LIN {X 0,Y 363.878,Z 264.828,A -85,B 0,C 180,E1 -13034.312,E2 -13034.312} C_VEL
LIN {X 0,Y 363.084,Z 274.413,A -85,B 0,C 180,E1 -13035.425,E2 -13035.425} C_VEL
LIN {X 0,Y 362.252,Z 284.208,A -85,B 0,C 180,E1 -13036.823,E2 -13036.823} C_VEL
LIN {X 0,Y 361.616,Z 292.231,A -85,B 0,C 180,E1 -13038.225,E2 -13038.225} C_VEL
LIN {X 0,Y 360.989,Z 300.051,A -85,B 0,C 180,E1 -13039.908,E2 -13039.908} C_VEL
LIN {X 0,Y 360.655,Z 306.321,A -85,B 0,C 180,E1 -13041.596,E2 -13041.596} C_VEL
LIN {X 0,Y 360.41,Z 311.284,A -85,B 0,C 180,E1 -13043.281,E2 -13043.281} C_VEL
LIN {X 0,Y 360.44,Z 315.106,A -85,B 0,C 180,E1 -13044.966,E2 -13044.966} C_VEL
LIN {X 0,Y 360.412,Z 317.873,A -85,B 0,C 180,E1 -13046.646,E2 -13046.646} C_VEL
LIN {X 0,Y 360.513,Z 319.178,A -85,B 0,C 180,E1 -13047.765,E2 -13047.765} C_VEL
LIN {X 0,Y 360.539,Z 320.076,A -85,B 0,C 180,E1 -13048.883,E2 -13048.883} C_VEL
LIN {X 0,Y 360.521,Z 320.55,A -85,B 0,C 180,E1 -13050,E2 -13050} C_VEL
LIN {X 0,Y 360.517,Z 320.6,A -85,B 0,C 180,E1 -13051.117,E2 -13051.117} C_VEL
LIN {X 0,Y 360.427,Z 320.257,A -85,B 0,C 180,E1 -13052.235,E2 -13052.235} C_VEL
LIN {X 0,Y 360.359,Z 319.529,A -85,B 0,C 180,E1 -13053.354,E2 -13053.354} C_VEL
LIN {X 0,Y 360.367,Z 318.397,A -85,B 0,C 180,E1 -13054.474,E2 -13054.474} C_VEL
LIN {X 0,Y 360.407,Z 314.826,A -85,B 0,C 180,E1 -13056.719,E2 -13056.719} C_VEL
LIN {X 0,Y 360.695,Z 310.995,A -85,B 0,C 180,E1 -13058.403,E2 -13058.403} C_VEL
LIN {X 0,Y 361.142,Z 306.058,A -85,B 0,C 180,E1 -13060.087,E2 -13060.087} C_VEL
LIN {X 0,Y 361.814,Z 299.872,A -85,B 0,C 180,E1 -13061.768,E2 -13061.768} C_VEL
LIN {X 0,Y 362.948,Z 292.218,A -85,B 0,C 180,E1 -13063.436,E2 -13063.436} C_VEL
LIN {X 0,Y 363.92,Z 283.963,A -85,B 0,C 180,E1 -13064.899,E2 -13064.899} C_VEL
LIN {X 0,Y 365.228,Z 273.856,A -85,B 0,C 180,E1 -13066.345,E2 -13066.345} C_VEL
LIN {X 0,Y 366.624,Z 263.144,A -85,B 0,C 180,E1 -13067.572,E2 -13067.572} C_VEL
LIN {X 0,Y 367.91,Z 252.779,A -85,B 0,C 180,E1 -13068.516,E2 -13068.516} C_VEL
LIN {X 0,Y 369.141,Z 240.378,A -85,B 0,C 180,E1 -13069.389,E2 -13069.389} C_VEL
LIN {X 0,Y 370.234,Z 227.35,A -85,B 0,C 180,E1 -13070.052,E2 -13070.052} C_VEL
LIN {X 0,Y 370.952,Z 214.539,A -85,B 0,C 180,E1 -13070.481,E2 -13070.481} C_VEL
LIN {X 0,Y 372.245,Z 144.582,A -85,B 0,C 180,E1 -13071.883,E2 -13071.883} C_VEL
LIN {X 0,Y 368.931,Z 123.307,A -85,B 0,C 180,E1 -13072.583,E2 -13072.583} C_VEL
LIN {X 0,Y 365.502,Z 106.451,A -85,B 0,C 180,E1 -13073.214,E2 -13073.214} C_VEL
LIN {X 0,Y 367.15,Z 91.794,A -85,B 0,C 180,E1 -13076.426,E2 -13076.426} C_VEL
LIN {X 0,Y 366.338,Z 86.268,A -85,B 0,C 180,E1 -13077.771,E2 -13077.771} C_VEL
LIN {X 0,Y 363.642,Z 74.544,A -85,B 0,C 180,E1 -13080.807,E2 -13080.807} C_VEL
LIN {X 0,Y 361.899,Z 67.405,A -85,B 0,C 180,E1 -13082.773,E2 -13082.773} C_VEL
LIN {X 0,Y 361.868,Z 67.406,A -85,B 0,C 180,E1 -13085.636,E2 -13085.636} C_VEL
LIN {X 0,Y 361.87,Z 67.408,A -85,B 0,C 180,E1 -13089.027,E2 -13089.027} C_VEL
LIN {X 0,Y 361.835,Z 67.413,A -85,B 0,C 180,E1 -13092.828,E2 -13092.828} C_VEL
LIN {X 0,Y 361.823,Z 67.401,A -85,B 0,C 180,E1 -13095.945,E2 -13095.945} C_VEL
LIN {X 0,Y 361.871,Z 67.406,A -85,B 0,C 180,E1 -13099.237,E2 -13099.237} C_VEL
LIN {X 0,Y 361.867,Z 67.405,A -85,B 0,C 180,E1 -13102.982,E2 -13102.982} C_VEL
LIN {X 0,Y 361.858,Z 67.407,A -85,B 0,C 180,E1 -13106.63,E2 -13106.63} C_VEL
LIN {X 0,Y 361.872,Z 67.404,A -85,B 0,C 180,E1 -13109.672,E2 -13109.672} C_VEL
LIN {X 0,Y 361.952,Z 67.392,A -85,B 0,C 180,E1 -13113.475,E2 -13113.475} C_VEL
LIN {X 0,Y 361.889,Z 67.397,A -85,B 0,C 180,E1 -13117.145,E2 -13117.145} C_VEL
LIN {X 0,Y 361.925,Z 67.399,A -85,B 0,C 180,E1 -13120.725,E2 -13120.725} C_VEL
LIN {X 0,Y 361.943,Z 67.399,A -85,B 0,C 180,E1 -13124.226,E2 -13124.226} C_VEL
LIN {X 0,Y 361.996,Z 67.384,A -85,B 0,C 180,E1 -13126.528,E2 -13126.528} C_VEL
LIN {X 0,Y 362.031,Z 67.39,A -85,B 0,C 180,E1 -13129.938,E2 -13129.938} C_VEL
LIN {X 0,Y 362.158,Z 67.365,A -85,B 0,C 180,E1 -13133.314,E2 -13133.314} C_VEL
LIN {X 0,Y 362.278,Z 67.349,A -85,B 0,C 180,E1 -13137.777,E2 -13137.777} C_VEL
LIN {X 0,Y 362.424,Z 67.341,A -85,B 0,C 180,E1 -13140,E2 -13140} C_VEL
LIN {X 0,Y 362.278,Z 67.348,A -85,B 0,C 180,E1 -13142.224,E2 -13142.224} C_VEL
LIN {X 0,Y 362.146,Z 67.372,A -85,B 0,C 180,E1 -13146.687,E2 -13146.687} C_VEL
LIN {X 0,Y 361.998,Z 67.392,A -85,B 0,C 180,E1 -13150.063,E2 -13150.063} C_VEL
LIN {X 0,Y 361.996,Z 67.389,A -85,B 0,C 180,E1 -13153.899,E2 -13153.899} C_VEL
LIN {X 0,Y 361.926,Z 67.397,A -85,B 0,C 180,E1 -13156.935,E2 -13156.935} C_VEL
LIN {X 0,Y 361.885,Z 67.408,A -85,B 0,C 180,E1 -13160.461,E2 -13160.461} C_VEL
LIN {X 0,Y 361.891,Z 67.406,A -85,B 0,C 180,E1 -13164.113,E2 -13164.113} C_VEL
LIN {X 0,Y 361.863,Z 67.409,A -85,B 0,C 180,E1 -13167.783,E2 -13167.783} C_VEL
LIN {X 0,Y 361.845,Z 67.411,A -85,B 0,C 180,E1 -13171.286,E2 -13171.286} C_VEL
LIN {X 0,Y 361.853,Z 67.412,A -85,B 0,C 180,E1 -13174.281,E2 -13174.281} C_VEL
LIN {X 0,Y 361.859,Z 67.41,A -85,B 0,C 180,E1 -13177.223,E2 -13177.223} C_VEL
LIN {X 0,Y 361.828,Z 67.405,A -85,B 0,C 180,E1 -13180.755,E2 -13180.755} C_VEL
LIN {X 0,Y 361.815,Z 67.414,A -85,B 0,C 180,E1 -13184.369,E2 -13184.369} C_VEL
LIN {X 0,Y 361.83,Z 67.418,A -85,B 0,C 180,E1 -13187.57,E2 -13187.57} C_VEL
LIN {X 0,Y 361.859,Z 67.492,A -85,B 0,C 180,E1 -13191.128,E2 -13191.128} C_VEL
LIN {X 0,Y 362.972,Z 72.191,A -85,B 0,C 180,E1 -13192.606,E2 -13192.606} C_VEL
LIN {X 0,Y 371.01,Z 90.504,A -85,B 0,C 180,E1 -13193.662,E2 -13193.662} C_VEL
LIN {X 0,Y 373.28,Z 96.119,A -85,B 0,C 180,E1 -13193.956,E2 -13193.956} C_VEL
LIN {X 0,Y 371.592,Z 178.35,A -85,B 0,C 180,E1 -13195.596,E2 -13195.596} C_VEL
LIN {X 0,Y 370.967,Z 191.99,A -85,B 0,C 180,E1 -13196.09,E2 -13196.09} C_VEL
LIN {X 0,Y 370.296,Z 204.055,A -85,B 0,C 180,E1 -13196.75,E2 -13196.75} C_VEL
LIN {X 0,Y 369.283,Z 216.174,A -85,B 0,C 180,E1 -13197.639,E2 -13197.639} C_VEL
LIN {X 0,Y 368.162,Z 226.889,A -85,B 0,C 180,E1 -13198.656,E2 -13198.656} C_VEL
LIN {X 0,Y 366.831,Z 237.592,A -85,B 0,C 180,E1 -13199.926,E2 -13199.926} C_VEL
LIN {X 0,Y 365.682,Z 246.772,A -85,B 0,C 180,E1 -13201.284,E2 -13201.284} C_VEL
LIN {X 0,Y 364.549,Z 254.831,A -85,B 0,C 180,E1 -13202.751,E2 -13202.751} C_VEL
LIN {X 0,Y 363.345,Z 262.608,A -85,B 0,C 180,E1 -13204.509,E2 -13204.509} C_VEL
LIN {X 0,Y 362.591,Z 267.841,A -85,B 0,C 180,E1 -13205.982,E2 -13205.982} C_VEL
LIN {X 0,Y 361.848,Z 272.838,A -85,B 0,C 180,E1 -13207.745,E2 -13207.745} C_VEL
LIN {X 0,Y 361.32,Z 276.612,A -85,B 0,C 180,E1 -13209.506,E2 -13209.506} C_VEL
LIN {X 0,Y 360.986,Z 278.531,A -85,B 0,C 180,E1 -13210.673,E2 -13210.673} C_VEL
LIN {X 0,Y 360.598,Z 280.76,A -85,B 0,C 180,E1 -13212.749,E2 -13212.749} C_VEL
LIN {X 0,Y 360.462,Z 281.512,A -85,B 0,C 180,E1 -13214.16,E2 -13214.16} C_VEL
LIN {X 0,Y 360.387,Z 281.658,A -85,B 0,C 180,E1 -13215.315,E2 -13215.315} C_VEL
LIN {X 0,Y 360.421,Z 281.016,A -85,B 0,C 180,E1 -13217.157,E2 -13217.157} C_VEL
LIN {X 0,Y 360.476,Z 279.603,A -85,B 0,C 180,E1 -13218.758,E2 -13218.758} C_VEL
LIN {X 0,Y 360.55,Z 278.064,A -85,B 0,C 180,E1 -13219.897,E2 -13219.897} C_VEL
LIN {X 0,Y 360.842,Z 274.948,A -85,B 0,C 180,E1 -13221.601,E2 -13221.601} C_VEL
LIN {X 0,Y 361.182,Z 270.774,A -85,B 0,C 180,E1 -13223.296,E2 -13223.296} C_VEL
LIN {X 0,Y 361.599,Z 264.43,A -85,B 0,C 180,E1 -13225.262,E2 -13225.262} C_VEL
LIN {X 0,Y 362.197,Z 257.516,A -85,B 0,C 180,E1 -13226.942,E2 -13226.942} C_VEL
LIN {X 0,Y 363.031,Z 248.837,A -85,B 0,C 180,E1 -13228.614,E2 -13228.614} C_VEL
LIN {X 0,Y 363.921,Z 239.937,A -85,B 0,C 180,E1 -13230,E2 -13230} C_VEL
LIN {X 0,Y 364.73,Z 230.191,A -85,B 0,C 180,E1 -13231.243,E2 -13231.243} C_VEL
LIN {X 0,Y 365.603,Z 219.374,A -85,B 0,C 180,E1 -13232.349,E2 -13232.349} C_VEL
LIN {X 0,Y 366.324,Z 207.473,A -85,B 0,C 180,E1 -13233.3,E2 -13233.3} C_VEL
LIN {X 0,Y 366.905,Z 194.367,A -85,B 0,C 180,E1 -13234.085,E2 -13234.085} C_VEL
LIN {X 0,Y 367.322,Z 181.85,A -85,B 0,C 180,E1 -13234.595,E2 -13234.595} C_VEL
LIN {X 0,Y 367.7,Z 164.255,A -85,B 0,C 180,E1 -13235.002,E2 -13235.002} C_VEL
LIN {X 0,Y 368.727,Z 93.086,A -85,B 0,C 180,E1 -13236.387,E2 -13236.387} C_VEL
LIN {X 0,Y 366.646,Z 83.395,A -85,B 0,C 180,E1 -13236.684,E2 -13236.684} C_VEL
LIN {X 0,Y 362.854,Z 71.16,A -85,B 0,C 180,E1 -13237.133,E2 -13237.133} C_VEL
LIN {X 0,Y 362.513,Z 69.324,A -85,B 0,C 180,E1 -13237.64,E2 -13237.64} C_VEL
LIN {X 0,Y 361.863,Z 68,A -85,B 0,C 180,E1 -13238.196,E2 -13238.196} C_VEL
LIN {X 0,Y 360.534,Z 67.575,A -85,B 0,C 180,E1 -13238.93,E2 -13238.93} C_VEL
LIN {X 0,Y 355.937,Z 68.203,A -85,B 0,C 180,E1 -13241.231,E2 -13241.231} C_VEL
LIN {X 0,Y 354.986,Z 68.271,A -85,B 0,C 180,E1 -13242.202,E2 -13242.202} C_VEL
LIN {X 0,Y 354.924,Z 68.276,A -85,B 0,C 180,E1 -13242.53,E2 -13242.53} C_VEL
LIN {X 0,Y 354.925,Z 68.272,A -85,B 0,C 180,E1 -13244.917,E2 -13244.917} C_VEL
LIN {X 0,Y 354.912,Z 68.277,A -85,B 0,C 180,E1 -13248.472,E2 -13248.472} C_VEL
LIN {X 0,Y 354.822,Z 68.289,A -85,B 0,C 180,E1 -13252.107,E2 -13252.107} C_VEL
LIN {X 0,Y 354.903,Z 68.277,A -85,B 0,C 180,E1 -13255.827,E2 -13255.827} C_VEL
LIN {X 0,Y 354.822,Z 68.287,A -85,B 0,C 180,E1 -13259.682,E2 -13259.682} C_VEL
LIN {X 0,Y 354.81,Z 68.29,A -85,B 0,C 180,E1 -13263.702,E2 -13263.702} C_VEL
LIN {X 0,Y 354.806,Z 68.286,A -85,B 0,C 180,E1 -13266.459,E2 -13266.459} C_VEL
LIN {X 0,Y 354.828,Z 68.287,A -85,B 0,C 180,E1 -13269.423,E2 -13269.423} C_VEL
LIN {X 0,Y 354.792,Z 68.288,A -85,B 0,C 180,E1 -13272.867,E2 -13272.867} C_VEL
LIN {X 0,Y 354.784,Z 68.289,A -85,B 0,C 180,E1 -13276.106,E2 -13276.106} C_VEL
LIN {X 0,Y 354.792,Z 68.293,A -85,B 0,C 180,E1 -13279.179,E2 -13279.179} C_VEL
LIN {X 0,Y 354.811,Z 68.285,A -85,B 0,C 180,E1 -13282.402,E2 -13282.402} C_VEL
LIN {X 0,Y 354.816,Z 68.29,A -85,B 0,C 180,E1 -13284.941,E2 -13284.941} C_VEL
LIN {X 0,Y 354.796,Z 68.288,A -85,B 0,C 180,E1 -13288.405,E2 -13288.405} C_VEL
LIN {X 0,Y 354.85,Z 68.28,A -85,B 0,C 180,E1 -13291.618,E2 -13291.618} C_VEL
LIN {X 0,Y 354.902,Z 68.275,A -85,B 0,C 180,E1 -13294.172,E2 -13294.172} C_VEL
LIN {X 0,Y 354.839,Z 68.282,A -85,B 0,C 180,E1 -13297.894,E2 -13297.894} C_VEL
LIN {X 0,Y 354.925,Z 68.272,A -85,B 0,C 180,E1 -13301.891,E2 -13301.891} C_VEL
LIN {X 0,Y 354.946,Z 68.271,A -85,B 0,C 180,E1 -13305.981,E2 -13305.981} C_VEL
LIN {X 0,Y 354.981,Z 68.266,A -85,B 0,C 180,E1 -13309.736,E2 -13309.736} C_VEL
LIN {X 0,Y 355.127,Z 68.246,A -85,B 0,C 180,E1 -13313.18,E2 -13313.18} C_VEL
LIN {X 0,Y 355.245,Z 68.236,A -85,B 0,C 180,E1 -13317.732,E2 -13317.732} C_VEL
LIN {X 0,Y 355.398,Z 68.216,A -85,B 0,C 180,E1 -13320,E2 -13320} C_VEL
LIN {X 0,Y 355.245,Z 68.232,A -85,B 0,C 180,E1 -13322.267,E2 -13322.267} C_VEL
LIN {X 0,Y 355.114,Z 68.248,A -85,B 0,C 180,E1 -13326.819,E2 -13326.819} C_VEL
LIN {X 0,Y 354.958,Z 68.267,A -85,B 0,C 180,E1 -13330.264,E2 -13330.264} C_VEL
LIN {X 0,Y 354.945,Z 68.269,A -85,B 0,C 180,E1 -13334.019,E2 -13334.019} C_VEL
LIN {X 0,Y 354.924,Z 68.271,A -85,B 0,C 180,E1 -13338.108,E2 -13338.108} C_VEL
LIN {X 0,Y 354.817,Z 68.284,A -85,B 0,C 180,E1 -13342.107,E2 -13342.107} C_VEL
LIN {X 0,Y 354.899,Z 68.274,A -85,B 0,C 180,E1 -13345.827,E2 -13345.827} C_VEL
LIN {X 0,Y 354.855,Z 68.279,A -85,B 0,C 180,E1 -13349.678,E2 -13349.678} C_VEL
LIN {X 0,Y 354.808,Z 68.285,A -85,B 0,C 180,E1 -13353.702,E2 -13353.702} C_VEL
LIN {X 0,Y 354.8,Z 68.292,A -85,B 0,C 180,E1 -13356.459,E2 -13356.459} C_VEL
LIN {X 0,Y 354.826,Z 68.283,A -85,B 0,C 180,E1 -13359.423,E2 -13359.423} C_VEL
LIN {X 0,Y 354.789,Z 68.289,A -85,B 0,C 180,E1 -13362.867,E2 -13362.867} C_VEL
LIN {X 0,Y 354.769,Z 68.296,A -85,B 0,C 180,E1 -13366.103,E2 -13366.103} C_VEL
LIN {X 0,Y 354.789,Z 68.288,A -85,B 0,C 180,E1 -13369.179,E2 -13369.179} C_VEL
LIN {X 0,Y 354.809,Z 68.287,A -85,B 0,C 180,E1 -13372.402,E2 -13372.402} C_VEL
LIN {X 0,Y 354.814,Z 68.285,A -85,B 0,C 180,E1 -13374.941,E2 -13374.941} C_VEL
LIN {X 0,Y 354.795,Z 68.288,A -85,B 0,C 180,E1 -13378.405,E2 -13378.405} C_VEL
LIN {X 0,Y 354.882,Z 68.376,A -85,B 0,C 180,E1 -13379.874,E2 -13379.874} C_VEL
LIN {X 0,Y 357.374,Z 80.376,A -85,B 0,C 180,E1 -13382.743,E2 -13382.743} C_VEL
LIN {X 0,Y 358.244,Z 86.354,A -85,B 0,C 180,E1 -13384.119,E2 -13384.119} C_VEL
LIN {X 0,Y 357.097,Z 100.352,A -85,B 0,C 180,E1 -13387.134,E2 -13387.134} C_VEL
LIN {X 0,Y 356.539,Z 106.915,A -85,B 0,C 180,E1 -13388.537,E2 -13388.537} C_VEL
LIN {X 0,Y 361.331,Z 145.067,A -85,B 0,C 180,E1 -13389.568,E2 -13389.568} C_VEL
LIN {X 0,Y 360.23,Z 215.998,A -85,B 0,C 180,E1 -13391,E2 -13391} C_VEL
LIN {X 0,Y 359.668,Z 229.27,A -85,B 0,C 180,E1 -13391.486,E2 -13391.486} C_VEL
LIN {X 0,Y 358.771,Z 242.008,A -85,B 0,C 180,E1 -13392.176,E2 -13392.176} C_VEL
LIN {X 0,Y 357.948,Z 253.353,A -85,B 0,C 180,E1 -13393.018,E2 -13393.018} C_VEL
LIN {X 0,Y 357.002,Z 263.768,A -85,B 0,C 180,E1 -13394.001,E2 -13394.001} C_VEL
LIN {X 0,Y 356.06,Z 274.562,A -85,B 0,C 180,E1 -13395.279,E2 -13395.279} C_VEL
LIN {X 0,Y 355.314,Z 283.359,A -85,B 0,C 180,E1 -13396.561,E2 -13396.561} C_VEL
LIN {X 0,Y 354.6,Z 291.455,A -85,B 0,C 180,E1 -13397.988,E2 -13397.988} C_VEL
LIN {X 0,Y 353.93,Z 299.371,A -85,B 0,C 180,E1 -13399.705,E2 -13399.705} C_VEL
LIN {X 0,Y 353.6,Z 305.7,A -85,B 0,C 180,E1 -13401.427,E2 -13401.427} C_VEL
LIN {X 0,Y 353.352,Z 310.715,A -85,B 0,C 180,E1 -13403.146,E2 -13403.146} C_VEL
LIN {X 0,Y 353.355,Z 314.584,A -85,B 0,C 180,E1 -13404.865,E2 -13404.865} C_VEL
LIN {X 0,Y 353.329,Z 317.395,A -85,B 0,C 180,E1 -13406.579,E2 -13406.579} C_VEL
LIN {X 0,Y 353.415,Z 318.72,A -85,B 0,C 180,E1 -13407.72,E2 -13407.72} C_VEL
LIN {X 0,Y 353.474,Z 319.641,A -85,B 0,C 180,E1 -13408.86,E2 -13408.86} C_VEL
LIN {X 0,Y 353.456,Z 320.152,A -85,B 0,C 180,E1 -13410,E2 -13410} C_VEL
LIN {X 0,Y 353.433,Z 320.225,A -85,B 0,C 180,E1 -13411.139,E2 -13411.139} C_VEL
LIN {X 0,Y 353.275,Z 319.194,A -85,B 0,C 180,E1 -13413.421,E2 -13413.421} C_VEL
LIN {X 0,Y 353.276,Z 318.094,A -85,B 0,C 180,E1 -13414.564,E2 -13414.564} C_VEL
LIN {X 0,Y 353.27,Z 316.242,A -85,B 0,C 180,E1 -13415.897,E2 -13415.897} C_VEL
LIN {X 0,Y 353.528,Z 312.18,A -85,B 0,C 180,E1 -13417.999,E2 -13417.999} C_VEL
LIN {X 0,Y 353.925,Z 307.672,A -85,B 0,C 180,E1 -13419.717,E2 -13419.717} C_VEL
LIN {X 0,Y 354.689,Z 300.891,A -85,B 0,C 180,E1 -13421.718,E2 -13421.718} C_VEL
LIN {X 0,Y 355.832,Z 293.54,A -85,B 0,C 180,E1 -13423.419,E2 -13423.419} C_VEL
LIN {X 0,Y 356.97,Z 284.618,A -85,B 0,C 180,E1 -13425.092,E2 -13425.092} C_VEL
LIN {X 0,Y 358.286,Z 275.092,A -85,B 0,C 180,E1 -13426.524,E2 -13426.524} C_VEL
LIN {X 0,Y 359.71,Z 264.725,A -85,B 0,C 180,E1 -13427.775,E2 -13427.775} C_VEL
LIN {X 0,Y 361.219,Z 253.242,A -85,B 0,C 180,E1 -13428.872,E2 -13428.872} C_VEL
LIN {X 0,Y 362.499,Z 241.208,A -85,B 0,C 180,E1 -13429.759,E2 -13429.759} C_VEL
LIN {X 0,Y 363.682,Z 227.862,A -85,B 0,C 180,E1 -13430.466,E2 -13430.466} C_VEL
LIN {X 0,Y 364.485,Z 214.443,A -85,B 0,C 180,E1 -13430.935,E2 -13430.935} C_VEL
LIN {X 0,Y 365.828,Z 145.241,A -85,B 0,C 180,E1 -13432.347,E2 -13432.347} C_VEL
LIN {X 0,Y 362.406,Z 123.714,A -85,B 0,C 180,E1 -13433.082,E2 -13433.082} C_VEL
LIN {X 0,Y 358.82,Z 106.008,A -85,B 0,C 180,E1 -13433.773,E2 -13433.773} C_VEL
LIN {X 0,Y 360.327,Z 93.124,A -85,B 0,C 180,E1 -13436.654,E2 -13436.654} C_VEL
LIN {X 0,Y 358.869,Z 85.019,A -85,B 0,C 180,E1 -13438.71,E2 -13438.71} C_VEL
LIN {X 0,Y 355.768,Z 71.967,A -85,B 0,C 180,E1 -13442.233,E2 -13442.233} C_VEL
LIN {X 0,Y 354.821,Z 68.289,A -85,B 0,C 180,E1 -13443.3,E2 -13443.3} C_VEL
LIN {X 0,Y 354.798,Z 68.292,A -85,B 0,C 180,E1 -13446.459,E2 -13446.459} C_VEL
LIN {X 0,Y 354.822,Z 68.288,A -85,B 0,C 180,E1 -13449.423,E2 -13449.423} C_VEL
LIN {X 0,Y 354.787,Z 68.291,A -85,B 0,C 180,E1 -13452.867,E2 -13452.867} C_VEL
LIN {X 0,Y 354.773,Z 68.28,A -85,B 0,C 180,E1 -13456.105,E2 -13456.105} C_VEL
LIN {X 0,Y 354.822,Z 68.284,A -85,B 0,C 180,E1 -13459.184,E2 -13459.184} C_VEL
LIN {X 0,Y 354.807,Z 68.282,A -85,B 0,C 180,E1 -13462.402,E2 -13462.402} C_VEL
LIN {X 0,Y 354.81,Z 68.287,A -85,B 0,C 180,E1 -13464.941,E2 -13464.941} C_VEL
LIN {X 0,Y 354.791,Z 68.29,A -85,B 0,C 180,E1 -13468.405,E2 -13468.405} C_VEL
LIN {X 0,Y 354.848,Z 68.282,A -85,B 0,C 180,E1 -13471.619,E2 -13471.619} C_VEL
LIN {X 0,Y 354.897,Z 68.272,A -85,B 0,C 180,E1 -13474.173,E2 -13474.173} C_VEL
LIN {X 0,Y 354.835,Z 68.274,A -85,B 0,C 180,E1 -13477.894,E2 -13477.894} C_VEL
LIN {X 0,Y 354.921,Z 68.266,A -85,B 0,C 180,E1 -13481.891,E2 -13481.891} C_VEL
LIN {X 0,Y 354.94,Z 68.269,A -85,B 0,C 180,E1 -13485.981,E2 -13485.981} C_VEL
LIN {X 0,Y 354.977,Z 68.267,A -85,B 0,C 180,E1 -13489.736,E2 -13489.736} C_VEL
LIN {X 0,Y 355.123,Z 68.241,A -85,B 0,C 180,E1 -13493.181,E2 -13493.181} C_VEL
LIN {X 0,Y 355.241,Z 68.225,A -85,B 0,C 180,E1 -13497.733,E2 -13497.733} C_VEL
LIN {X 0,Y 355.393,Z 68.217,A -85,B 0,C 180,E1 -13500,E2 -13500} C_VEL
LIN {X 0,Y 355.241,Z 68.224,A -85,B 0,C 180,E1 -13502.268,E2 -13502.268} C_VEL
LIN {X 0,Y 355.109,Z 68.249,A -85,B 0,C 180,E1 -13506.82,E2 -13506.82} C_VEL
LIN {X 0,Y 354.954,Z 68.269,A -85,B 0,C 180,E1 -13510.265,E2 -13510.265} C_VEL
LIN {X 0,Y 354.941,Z 68.268,A -85,B 0,C 180,E1 -13514.019,E2 -13514.019} C_VEL
LIN {X 0,Y 354.888,Z 68.271,A -85,B 0,C 180,E1 -13518.093,E2 -13518.093} C_VEL
LIN {X 0,Y 354.817,Z 68.279,A -85,B 0,C 180,E1 -13521.419,E2 -13521.419} C_VEL
LIN {X 0,Y 354.852,Z 68.283,A -85,B 0,C 180,E1 -13524.577,E2 -13524.577} C_VEL
LIN {X 0,Y 354.808,Z 68.288,A -85,B 0,C 180,E1 -13528.385,E2 -13528.385} C_VEL
LIN {X 0,Y 354.786,Z 68.289,A -85,B 0,C 180,E1 -13532.334,E2 -13532.334} C_VEL
LIN {X 0,Y 354.821,Z 68.283,A -85,B 0,C 180,E1 -13535.7,E2 -13535.7} C_VEL
LIN {X 0,Y 354.798,Z 68.293,A -85,B 0,C 180,E1 -13539.419,E2 -13539.419} C_VEL
LIN {X 0,Y 354.785,Z 68.297,A -85,B 0,C 180,E1 -13542.867,E2 -13542.867} C_VEL
LIN {X 0,Y 354.766,Z 68.296,A -85,B 0,C 180,E1 -13546.104,E2 -13546.104} C_VEL
LIN {X 0,Y 354.765,Z 68.295,A -85,B 0,C 180,E1 -13549.177,E2 -13549.177} C_VEL
LIN {X 0,Y 354.816,Z 68.461,A -85,B 0,C 180,E1 -13550.667,E2 -13550.667} C_VEL
LIN {X 0,Y 355.816,Z 72.665,A -85,B 0,C 180,E1 -13552.016,E2 -13552.016} C_VEL
LIN {X 0,Y 364.858,Z 92.844,A -85,B 0,C 180,E1 -13553.226,E2 -13553.226} C_VEL
LIN {X 0,Y 366.995,Z 98.441,A -85,B 0,C 180,E1 -13553.518,E2 -13553.518} C_VEL
LIN {X 0,Y 365.147,Z 179.189,A -85,B 0,C 180,E1 -13555.153,E2 -13555.153} C_VEL
LIN {X 0,Y 364.478,Z 192.945,A -85,B 0,C 180,E1 -13555.667,E2 -13555.667} C_VEL
LIN {X 0,Y 363.747,Z 205.328,A -85,B 0,C 180,E1 -13556.367,E2 -13556.367} C_VEL
LIN {X 0,Y 362.628,Z 217.542,A -85,B 0,C 180,E1 -13557.301,E2 -13557.301} C_VEL
LIN {X 0,Y 361.462,Z 228.075,A -85,B 0,C 180,E1 -13558.334,E2 -13558.334} C_VEL
LIN {X 0,Y 360.035,Z 238.914,A -85,B 0,C 180,E1 -13559.663,E2 -13559.663} C_VEL
LIN {X 0,Y 358.88,Z 247.664,A -85,B 0,C 180,E1 -13561.009,E2 -13561.009} C_VEL
LIN {X 0,Y 357.64,Z 255.855,A -85,B 0,C 180,E1 -13562.551,E2 -13562.551} C_VEL
LIN {X 0,Y 356.435,Z 263.319,A -85,B 0,C 180,E1 -13564.293,E2 -13564.293} C_VEL
LIN {X 0,Y 355.479,Z 269.421,A -85,B 0,C 180,E1 -13566.091,E2 -13566.091} C_VEL
LIN {X 0,Y 354.744,Z 274.153,A -85,B 0,C 180,E1 -13567.889,E2 -13567.889} C_VEL
LIN {X 0,Y 354.382,Z 276.606,A -85,B 0,C 180,E1 -13569.086,E2 -13569.086} C_VEL
LIN {X 0,Y 354.004,Z 278.592,A -85,B 0,C 180,E1 -13570.276,E2 -13570.276} C_VEL
LIN {X 0,Y 353.755,Z 280.127,A -85,B 0,C 180,E1 -13571.466,E2 -13571.466} C_VEL
LIN {X 0,Y 353.539,Z 281.176,A -85,B 0,C 180,E1 -13572.652,E2 -13572.652} C_VEL
LIN {X 0,Y 353.408,Z 281.814,A -85,B 0,C 180,E1 -13573.835,E2 -13573.835} C_VEL
LIN {X 0,Y 353.329,Z 282.052,A -85,B 0,C 180,E1 -13575.015,E2 -13575.015} C_VEL
LIN {X 0,Y 353.342,Z 281.431,A -85,B 0,C 180,E1 -13577.065,E2 -13577.065} C_VEL
LIN {X 0,Y 353.39,Z 280.199,A -85,B 0,C 180,E1 -13578.529,E2 -13578.529} C_VEL
LIN {X 0,Y 353.437,Z 278.774,A -85,B 0,C 180,E1 -13579.691,E2 -13579.691} C_VEL
LIN {X 0,Y 353.736,Z 275.777,A -85,B 0,C 180,E1 -13581.431,E2 -13581.431} C_VEL
LIN {X 0,Y 354.081,Z 271.736,A -85,B 0,C 180,E1 -13583.161,E2 -13583.161} C_VEL
LIN {X 0,Y 354.495,Z 265.54,A -85,B 0,C 180,E1 -13585.167,E2 -13585.167} C_VEL
LIN {X 0,Y 355.089,Z 258.789,A -85,B 0,C 180,E1 -13586.88,E2 -13586.88} C_VEL
LIN {X 0,Y 355.939,Z 250.388,A -85,B 0,C 180,E1 -13588.586,E2 -13588.586} C_VEL
LIN {X 0,Y 356.795,Z 241.73,A -85,B 0,C 180,E1 -13590,E2 -13590} C_VEL
LIN {X 0,Y 357.743,Z 231.09,A -85,B 0,C 180,E1 -13591.408,E2 -13591.408} C_VEL
LIN {X 0,Y 358.694,Z 220.019,A -85,B 0,C 180,E1 -13592.572,E2 -13592.572} C_VEL
LIN {X 0,Y 359.412,Z 208.174,A -85,B 0,C 180,E1 -13593.543,E2 -13593.543} C_VEL
LIN {X 0,Y 360.046,Z 194.964,A -85,B 0,C 180,E1 -13594.353,E2 -13594.353} C_VEL
LIN {X 0,Y 360.48,Z 181.966,A -85,B 0,C 180,E1 -13594.893,E2 -13594.893} C_VEL
LIN {X 0,Y 360.875,Z 164.179,A -85,B 0,C 180,E1 -13595.308,E2 -13595.308} C_VEL
LIN {X 0,Y 361.903,Z 93.961,A -85,B 0,C 180,E1 -13596.701,E2 -13596.701} C_VEL
LIN {X 0,Y 359.981,Z 85.067,A -85,B 0,C 180,E1 -13596.981,E2 -13596.981} C_VEL
LIN {X 0,Y 355.719,Z 71.491,A -85,B 0,C 180,E1 -13597.504,E2 -13597.504} C_VEL
LIN {X 0,Y 355.112,Z 68.253,A -85,B 0,C 180,E1 -13598.444,E2 -13598.444} C_VEL
LIN {X 0,Y 354.924,Z 68.276,A -85,B 0,C 180,E1 -13602.53,E2 -13602.53} C_VEL
LIN {X 0,Y 354.278,Z 68.363,A -85,B 0,C 180,E1 -13603.477,E2 -13603.477} C_VEL
LIN {X 0,Y 351.382,Z 68.721,A -85,B 0,C 180,E1 -13605.015,E2 -13605.015} C_VEL
LIN {X 0,Y 348.937,Z 69.022,A -85,B 0,C 180,E1 -13606.261,E2 -13606.261} C_VEL
LIN {X 0,Y 347.925,Z 69.143,A -85,B 0,C 180,E1 -13607.225,E2 -13607.225} C_VEL
LIN {X 0,Y 347.864,Z 69.151,A -85,B 0,C 180,E1 -13607.552,E2 -13607.552} C_VEL
LIN {X 0,Y 347.786,Z 69.16,A -85,B 0,C 180,E1 -13611.331,E2 -13611.331} C_VEL
LIN {X 0,Y 347.816,Z 69.156,A -85,B 0,C 180,E1 -13615.109,E2 -13615.109} C_VEL
LIN {X 0,Y 347.813,Z 69.16,A -85,B 0,C 180,E1 -13617.694,E2 -13617.694} C_VEL
LIN {X 0,Y 347.754,Z 69.166,A -85,B 0,C 180,E1 -13620.348,E2 -13620.348} C_VEL
LIN {X 0,Y 347.753,Z 69.167,A -85,B 0,C 180,E1 -13624.044,E2 -13624.044} C_VEL
LIN {X 0,Y 347.77,Z 69.165,A -85,B 0,C 180,E1 -13627.32,E2 -13627.32} C_VEL
LIN {X 0,Y 347.737,Z 69.167,A -85,B 0,C 180,E1 -13630.297,E2 -13630.297} C_VEL
LIN {X 0,Y 347.727,Z 69.173,A -85,B 0,C 180,E1 -13633.408,E2 -13633.408} C_VEL
LIN {X 0,Y 347.731,Z 69.168,A -85,B 0,C 180,E1 -13636.686,E2 -13636.686} C_VEL
LIN {X 0,Y 347.751,Z 69.164,A -85,B 0,C 180,E1 -13640.173,E2 -13640.173} C_VEL
LIN {X 0,Y 347.765,Z 69.165,A -85,B 0,C 180,E1 -13642.679,E2 -13642.679} C_VEL
LIN {X 0,Y 347.752,Z 69.164,A -85,B 0,C 180,E1 -13645.956,E2 -13645.956} C_VEL
LIN {X 0,Y 347.753,Z 69.164,A -85,B 0,C 180,E1 -13649.652,E2 -13649.652} C_VEL
LIN {X 0,Y 347.834,Z 69.154,A -85,B 0,C 180,E1 -13653.607,E2 -13653.607} C_VEL
LIN {X 0,Y 347.793,Z 69.161,A -85,B 0,C 180,E1 -13656.162,E2 -13656.162} C_VEL
LIN {X 0,Y 347.816,Z 69.157,A -85,B 0,C 180,E1 -13659.909,E2 -13659.909} C_VEL
LIN {X 0,Y 347.869,Z 69.155,A -85,B 0,C 180,E1 -13662.359,E2 -13662.359} C_VEL
LIN {X 0,Y 347.9,Z 69.149,A -85,B 0,C 180,E1 -13665.971,E2 -13665.971} C_VEL
LIN {X 0,Y 347.931,Z 69.143,A -85,B 0,C 180,E1 -13669.525,E2 -13669.525} C_VEL
LIN {X 0,Y 348.093,Z 69.122,A -85,B 0,C 180,E1 -13673.042,E2 -13673.042} C_VEL
LIN {X 0,Y 348.208,Z 69.112,A -85,B 0,C 180,E1 -13677.686,E2 -13677.686} C_VEL
LIN {X 0,Y 348.347,Z 69.094,A -85,B 0,C 180,E1 -13680,E2 -13680} C_VEL
LIN {X 0,Y 348.208,Z 69.108,A -85,B 0,C 180,E1 -13682.313,E2 -13682.313} C_VEL
LIN {X 0,Y 348.079,Z 69.125,A -85,B 0,C 180,E1 -13686.958,E2 -13686.958} C_VEL
LIN {X 0,Y 347.899,Z 69.146,A -85,B 0,C 180,E1 -13690.475,E2 -13690.475} C_VEL
LIN {X 0,Y 347.901,Z 69.146,A -85,B 0,C 180,E1 -13694.15,E2 -13694.15} C_VEL
LIN {X 0,Y 347.893,Z 69.147,A -85,B 0,C 180,E1 -13698.29,E2 -13698.29} C_VEL
LIN {X 0,Y 347.769,Z 69.163,A -85,B 0,C 180,E1 -13701.626,E2 -13701.626} C_VEL
LIN {X 0,Y 347.813,Z 69.161,A -85,B 0,C 180,E1 -13705.108,E2 -13705.108} C_VEL
LIN {X 0,Y 347.811,Z 69.157,A -85,B 0,C 180,E1 -13707.694,E2 -13707.694} C_VEL
LIN {X 0,Y 347.766,Z 69.165,A -85,B 0,C 180,E1 -13710.346,E2 -13710.346} C_VEL
LIN {X 0,Y 347.746,Z 69.17,A -85,B 0,C 180,E1 -13714.464,E2 -13714.464} C_VEL
LIN {X 0,Y 347.775,Z 69.163,A -85,B 0,C 180,E1 -13717.988,E2 -13717.988} C_VEL
LIN {X 0,Y 347.752,Z 69.166,A -85,B 0,C 180,E1 -13721.83,E2 -13721.83} C_VEL
LIN {X 0,Y 347.707,Z 69.17,A -85,B 0,C 180,E1 -13725.026,E2 -13725.026} C_VEL
LIN {X 0,Y 347.752,Z 69.167,A -85,B 0,C 180,E1 -13728.397,E2 -13728.397} C_VEL
LIN {X 0,Y 347.775,Z 69.167,A -85,B 0,C 180,E1 -13732.011,E2 -13732.011} C_VEL
LIN {X 0,Y 347.746,Z 69.168,A -85,B 0,C 180,E1 -13735.536,E2 -13735.536} C_VEL
LIN {X 0,Y 347.848,Z 69.323,A -85,B 0,C 180,E1 -13739.619,E2 -13739.619} C_VEL
LIN {X 0,Y 350.306,Z 81.191,A -85,B 0,C 180,E1 -13742.52,E2 -13742.52} C_VEL
LIN {X 0,Y 351.24,Z 86.967,A -85,B 0,C 180,E1 -13743.883,E2 -13743.883} C_VEL
LIN {X 0,Y 350.393,Z 98.157,A -85,B 0,C 180,E1 -13746.35,E2 -13746.35} C_VEL
LIN {X 0,Y 349.601,Z 106.602,A -85,B 0,C 180,E1 -13748.191,E2 -13748.191} C_VEL
LIN {X 0,Y 354.508,Z 145.666,A -85,B 0,C 180,E1 -13749.259,E2 -13749.259} C_VEL
LIN {X 0,Y 353.401,Z 215.496,A -85,B 0,C 180,E1 -13750.693,E2 -13750.693} C_VEL
LIN {X 0,Y 352.853,Z 228.044,A -85,B 0,C 180,E1 -13751.153,E2 -13751.153} C_VEL
LIN {X 0,Y 351.892,Z 241.574,A -85,B 0,C 180,E1 -13751.891,E2 -13751.891} C_VEL
LIN {X 0,Y 350.978,Z 253.74,A -85,B 0,C 180,E1 -13752.821,E2 -13752.821} C_VEL
LIN {X 0,Y 350.011,Z 264.014,A -85,B 0,C 180,E1 -13753.823,E2 -13753.823} C_VEL
LIN {X 0,Y 349.011,Z 274.84,A -85,B 0,C 180,E1 -13755.144,E2 -13755.144} C_VEL
LIN {X 0,Y 348.169,Z 284.302,A -85,B 0,C 180,E1 -13756.577,E2 -13756.577} C_VEL
LIN {X 0,Y 347.358,Z 293.536,A -85,B 0,C 180,E1 -13758.327,E2 -13758.327} C_VEL
LIN {X 0,Y 346.753,Z 300.964,A -85,B 0,C 180,E1 -13760.079,E2 -13760.079} C_VEL
LIN {X 0,Y 346.46,Z 306.918,A -85,B 0,C 180,E1 -13761.836,E2 -13761.836} C_VEL
LIN {X 0,Y 346.238,Z 311.727,A -85,B 0,C 180,E1 -13763.648,E2 -13763.648} C_VEL
LIN {X 0,Y 346.302,Z 315.14,A -85,B 0,C 180,E1 -13765.343,E2 -13765.343} C_VEL
LIN {X 0,Y 346.249,Z 316.917,A -85,B 0,C 180,E1 -13766.509,E2 -13766.509} C_VEL
LIN {X 0,Y 346.317,Z 318.262,A -85,B 0,C 180,E1 -13767.673,E2 -13767.673} C_VEL
LIN {X 0,Y 346.41,Z 319.206,A -85,B 0,C 180,E1 -13768.837,E2 -13768.837} C_VEL
LIN {X 0,Y 346.392,Z 319.746,A -85,B 0,C 180,E1 -13770,E2 -13770} C_VEL
LIN {X 0,Y 346.35,Z 319.849,A -85,B 0,C 180,E1 -13771.162,E2 -13771.162} C_VEL
LIN {X 0,Y 346.193,Z 318.858,A -85,B 0,C 180,E1 -13773.491,E2 -13773.491} C_VEL
LIN {X 0,Y 346.188,Z 317.783,A -85,B 0,C 180,E1 -13774.657,E2 -13774.657} C_VEL
LIN {X 0,Y 346.197,Z 316.178,A -85,B 0,C 180,E1 -13775.884,E2 -13775.884} C_VEL
LIN {X 0,Y 346.48,Z 311.951,A -85,B 0,C 180,E1 -13778.162,E2 -13778.162} C_VEL
LIN {X 0,Y 346.894,Z 307.492,A -85,B 0,C 180,E1 -13779.916,E2 -13779.916} C_VEL
LIN {X 0,Y 347.709,Z 300.798,A -85,B 0,C 180,E1 -13781.956,E2 -13781.956} C_VEL
LIN {X 0,Y 348.911,Z 293.517,A -85,B 0,C 180,E1 -13783.69,E2 -13783.69} C_VEL
LIN {X 0,Y 350.02,Z 285.272,A -85,B 0,C 180,E1 -13785.291,E2 -13785.291} C_VEL
LIN {X 0,Y 351.478,Z 275.287,A -85,B 0,C 180,E1 -13786.854,E2 -13786.854} C_VEL
LIN {X 0,Y 352.982,Z 265.045,A -85,B 0,C 180,E1 -13788.125,E2 -13788.125} C_VEL
LIN {X 0,Y 354.526,Z 253.723,A -85,B 0,C 180,E1 -13789.242,E2 -13789.242} C_VEL
LIN {X 0,Y 355.866,Z 241.993,A -85,B 0,C 180,E1 -13790.143,E2 -13790.143} C_VEL
LIN {X 0,Y 357.074,Z 229.144,A -85,B 0,C 180,E1 -13790.862,E2 -13790.862} C_VEL
LIN {X 0,Y 358,Z 215.468,A -85,B 0,C 180,E1 -13791.371,E2 -13791.371} C_VEL
LIN {X 0,Y 359.49,Z 146.357,A -85,B 0,C 180,E1 -13792.814,E2 -13792.814} C_VEL
LIN {X 0,Y 355.918,Z 124.025,A -85,B 0,C 180,E1 -13793.602,E2 -13793.602} C_VEL
LIN {X 0,Y 352.14,Z 105.526,A -85,B 0,C 180,E1 -13794.364,E2 -13794.364} C_VEL
LIN {X 0,Y 353.472,Z 95.117,A -85,B 0,C 180,E1 -13796.739,E2 -13796.739} C_VEL
LIN {X 0,Y 352.461,Z 88.724,A -85,B 0,C 180,E1 -13798.377,E2 -13798.377} C_VEL
LIN {X 0,Y 349.795,Z 77.298,A -85,B 0,C 180,E1 -13801.492,E2 -13801.492} C_VEL
LIN {X 0,Y 347.771,Z 69.172,A -85,B 0,C 180,E1 -13803.83,E2 -13803.83} C_VEL
LIN {X 0,Y 347.762,Z 69.166,A -85,B 0,C 180,E1 -13807.32,E2 -13807.32} C_VEL
LIN {X 0,Y 347.731,Z 69.17,A -85,B 0,C 180,E1 -13810.296,E2 -13810.296} C_VEL
LIN {X 0,Y 347.721,Z 69.174,A -85,B 0,C 180,E1 -13813.408,E2 -13813.408} C_VEL
LIN {X 0,Y 347.744,Z 69.161,A -85,B 0,C 180,E1 -13816.682,E2 -13816.682} C_VEL
LIN {X 0,Y 347.756,Z 69.166,A -85,B 0,C 180,E1 -13820.171,E2 -13820.171} C_VEL
LIN {X 0,Y 347.769,Z 69.165,A -85,B 0,C 180,E1 -13823.934,E2 -13823.934} C_VEL
LIN {X 0,Y 347.74,Z 69.168,A -85,B 0,C 180,E1 -13826.929,E2 -13826.929} C_VEL
LIN {X 0,Y 347.803,Z 69.163,A -85,B 0,C 180,E1 -13830.99,E2 -13830.99} C_VEL
LIN {X 0,Y 347.829,Z 69.151,A -85,B 0,C 180,E1 -13833.608,E2 -13833.608} C_VEL
LIN {X 0,Y 347.786,Z 69.162,A -85,B 0,C 180,E1 -13836.162,E2 -13836.162} C_VEL
LIN {X 0,Y 347.825,Z 69.157,A -85,B 0,C 180,E1 -13839.91,E2 -13839.91} C_VEL
LIN {X 0,Y 347.864,Z 69.144,A -85,B 0,C 180,E1 -13842.359,E2 -13842.359} C_VEL
LIN {X 0,Y 347.895,Z 69.147,A -85,B 0,C 180,E1 -13845.971,E2 -13845.971} C_VEL
LIN {X 0,Y 347.927,Z 69.144,A -85,B 0,C 180,E1 -13849.526,E2 -13849.526} C_VEL
LIN {X 0,Y 348.089,Z 69.117,A -85,B 0,C 180,E1 -13853.042,E2 -13853.042} C_VEL
LIN {X 0,Y 348.203,Z 69.101,A -85,B 0,C 180,E1 -13857.687,E2 -13857.687} C_VEL
LIN {X 0,Y 348.342,Z 69.095,A -85,B 0,C 180,E1 -13860,E2 -13860} C_VEL
LIN {X 0,Y 348.203,Z 69.1,A -85,B 0,C 180,E1 -13862.314,E2 -13862.314} C_VEL
LIN {X 0,Y 348.075,Z 69.124,A -85,B 0,C 180,E1 -13866.959,E2 -13866.959} C_VEL
LIN {X 0,Y 347.894,Z 69.148,A -85,B 0,C 180,E1 -13870.476,E2 -13870.476} C_VEL
LIN {X 0,Y 347.896,Z 69.145,A -85,B 0,C 180,E1 -13874.15,E2 -13874.15} C_VEL
LIN {X 0,Y 347.827,Z 69.151,A -85,B 0,C 180,E1 -13878.26,E2 -13878.26} C_VEL
LIN {X 0,Y 347.766,Z 69.156,A -85,B 0,C 180,E1 -13881.627,E2 -13881.627} C_VEL
LIN {X 0,Y 347.791,Z 69.156,A -85,B 0,C 180,E1 -13885.111,E2 -13885.111} C_VEL
LIN {X 0,Y 347.755,Z 69.161,A -85,B 0,C 180,E1 -13889.015,E2 -13889.015} C_VEL
LIN {X 0,Y 347.732,Z 69.169,A -85,B 0,C 180,E1 -13893.073,E2 -13893.073} C_VEL
LIN {X 0,Y 347.769,Z 69.165,A -85,B 0,C 180,E1 -13896.066,E2 -13896.066} C_VEL
LIN {X 0,Y 347.73,Z 69.174,A -85,B 0,C 180,E1 -13898.796,E2 -13898.796} C_VEL
LIN {X 0,Y 347.746,Z 69.161,A -85,B 0,C 180,E1 -13901.832,E2 -13901.832} C_VEL
LIN {X 0,Y 347.704,Z 69.169,A -85,B 0,C 180,E1 -13905.028,E2 -13905.028} C_VEL
LIN {X 0,Y 347.741,Z 69.171,A -85,B 0,C 180,E1 -13908.4,E2 -13908.4} C_VEL
LIN {X 0,Y 347.721,Z 69.219,A -85,B 0,C 180,E1 -13910.1,E2 -13910.1} C_VEL
LIN {X 0,Y 348.694,Z 73.239,A -85,B 0,C 180,E1 -13911.389,E2 -13911.389} C_VEL
LIN {X 0,Y 357.548,Z 92.446,A -85,B 0,C 180,E1 -13912.612,E2 -13912.612} C_VEL
LIN {X 0,Y 360.625,Z 99.914,A -85,B 0,C 180,E1 -13913.038,E2 -13913.038} C_VEL
LIN {X 0,Y 358.776,Z 178.778,A -85,B 0,C 180,E1 -13914.657,E2 -13914.657} C_VEL
LIN {X 0,Y 358.092,Z 192.005,A -85,B 0,C 180,E1 -13915.138,E2 -13915.138} C_VEL
LIN {X 0,Y 357.354,Z 204.58,A -85,B 0,C 180,E1 -13915.841,E2 -13915.841} C_VEL
LIN {X 0,Y 356.356,Z 215.514,A -85,B 0,C 180,E1 -13916.651,E2 -13916.651} C_VEL
LIN {X 0,Y 355.101,Z 226.551,A -85,B 0,C 180,E1 -13917.699,E2 -13917.699} C_VEL
LIN {X 0,Y 353.619,Z 237.731,A -85,B 0,C 180,E1 -13919.053,E2 -13919.053} C_VEL
LIN {X 0,Y 352.27,Z 246.764,A -85,B 0,C 180,E1 -13920.411,E2 -13920.411} C_VEL
LIN {X 0,Y 350.923,Z 255.815,A -85,B 0,C 180,E1 -13922.11,E2 -13922.11} C_VEL
LIN {X 0,Y 349.706,Z 262.89,A -85,B 0,C 180,E1 -13923.761,E2 -13923.761} C_VEL
LIN {X 0,Y 348.667,Z 269.178,A -85,B 0,C 180,E1 -13925.603,E2 -13925.603} C_VEL
LIN {X 0,Y 347.838,Z 274.028,A -85,B 0,C 180,E1 -13927.426,E2 -13927.426} C_VEL
LIN {X 0,Y 347.251,Z 277.694,A -85,B 0,C 180,E1 -13929.257,E2 -13929.257} C_VEL
LIN {X 0,Y 346.76,Z 280.263,A -85,B 0,C 180,E1 -13931.078,E2 -13931.078} C_VEL
LIN {X 0,Y 346.479,Z 281.517,A -85,B 0,C 180,E1 -13932.432,E2 -13932.432} C_VEL
LIN {X 0,Y 346.249,Z 282.414,A -85,B 0,C 180,E1 -13934.701,E2 -13934.701} C_VEL
LIN {X 0,Y 346.269,Z 281.848,A -85,B 0,C 180,E1 -13936.966,E2 -13936.966} C_VEL
LIN {X 0,Y 346.279,Z 280.794,A -85,B 0,C 180,E1 -13938.291,E2 -13938.291} C_VEL
LIN {X 0,Y 346.328,Z 279.437,A -85,B 0,C 180,E1 -13939.477,E2 -13939.477} C_VEL
LIN {X 0,Y 346.615,Z 276.557,A -85,B 0,C 180,E1 -13941.254,E2 -13941.254} C_VEL
LIN {X 0,Y 346.947,Z 272.647,A -85,B 0,C 180,E1 -13943.019,E2 -13943.019} C_VEL
LIN {X 0,Y 347.294,Z 267.616,A -85,B 0,C 180,E1 -13944.776,E2 -13944.776} C_VEL
LIN {X 0,Y 347.859,Z 261.286,A -85,B 0,C 180,E1 -13946.526,E2 -13946.526} C_VEL
LIN {X 0,Y 348.703,Z 253.338,A -85,B 0,C 180,E1 -13948.268,E2 -13948.268} C_VEL
LIN {X 0,Y 349.494,Z 245.258,A -85,B 0,C 180,E1 -13949.712,E2 -13949.712} C_VEL
LIN {X 0,Y 350.475,Z 235.394,A -85,B 0,C 180,E1 -13951.149,E2 -13951.149} C_VEL
LIN {X 0,Y 351.333,Z 225.708,A -85,B 0,C 180,E1 -13952.293,E2 -13952.293} C_VEL
LIN {X 0,Y 352.272,Z 213.486,A -85,B 0,C 180,E1 -13953.432,E2 -13953.432} C_VEL
LIN {X 0,Y 352.987,Z 200.862,A -85,B 0,C 180,E1 -13954.328,E2 -13954.328} C_VEL
LIN {X 0,Y 353.489,Z 187.717,A -85,B 0,C 180,E1 -13954.99,E2 -13954.99} C_VEL
LIN {X 0,Y 353.896,Z 174.188,A -85,B 0,C 180,E1 -13955.413,E2 -13955.413} C_VEL
LIN {X 0,Y 355.227,Z 95.348,A -85,B 0,C 180,E1 -13957.005,E2 -13957.005} C_VEL
LIN {X 0,Y 353.361,Z 86.985,A -85,B 0,C 180,E1 -13957.277,E2 -13957.277} C_VEL
LIN {X 0,Y 348.591,Z 71.835,A -85,B 0,C 180,E1 -13957.881,E2 -13957.881} C_VEL
LIN {X 0,Y 348.023,Z 69.136,A -85,B 0,C 180,E1 -13958.727,E2 -13958.727} C_VEL
LIN {X 0,Y 347.895,Z 69.149,A -85,B 0,C 180,E1 -13962.84,E2 -13962.84} C_VEL
LIN {X 0,Y 347.845,Z 69.158,A -85,B 0,C 180,E1 -13966.431,E2 -13966.431} C_VEL
LIN {X 0,Y 347.864,Z 69.151,A -85,B 0,C 180,E1 -13967.552,E2 -13967.552} C_VEL
LIN {X 0,Y 347.236,Z 69.233,A -85,B 0,C 180,E1 -13968.518,E2 -13968.518} C_VEL
LIN {X 0,Y 344.328,Z 69.595,A -85,B 0,C 180,E1 -13970.087,E2 -13970.087} C_VEL
LIN {X 0,Y 341.84,Z 69.902,A -85,B 0,C 180,E1 -13971.357,E2 -13971.357} C_VEL
LIN {X 0,Y 340.785,Z 70.036,A -85,B 0,C 180,E1 -13972.342,E2 -13972.342} C_VEL
LIN {X 0,Y 340.708,Z 70.04,A -85,B 0,C 180,E1 -13972.676,E2 -13972.676} C_VEL
LIN {X 0,Y 340.777,Z 70.036,A -85,B 0,C 180,E1 -13975.664,E2 -13975.664} C_VEL
LIN {X 0,Y 340.733,Z 70.041,A -85,B 0,C 180,E1 -13978.321,E2 -13978.321} C_VEL
LIN {X 0,Y 340.703,Z 70.043,A -85,B 0,C 180,E1 -13981.045,E2 -13981.045} C_VEL
LIN {X 0,Y 340.723,Z 70.042,A -85,B 0,C 180,E1 -13985.279,E2 -13985.279} C_VEL
LIN {X 0,Y 340.716,Z 70.041,A -85,B 0,C 180,E1 -13988.386,E2 -13988.386} C_VEL
LIN {X 0,Y 340.703,Z 70.044,A -85,B 0,C 180,E1 -13992.045,E2 -13992.045} C_VEL
LIN {X 0,Y 340.688,Z 70.049,A -85,B 0,C 180,E1 -13995.461,E2 -13995.461} C_VEL
LIN {X 0,Y 340.69,Z 70.045,A -85,B 0,C 180,E1 -13998.69,E2 -13998.69} C_VEL
LIN {X 0,Y 340.737,Z 70.038,A -85,B 0,C 180,E1 -14001.772,E2 -14001.772} C_VEL
LIN {X 0,Y 340.726,Z 70.04,A -85,B 0,C 180,E1 -14005.595,E2 -14005.595} C_VEL
LIN {X 0,Y 340.701,Z 70.048,A -85,B 0,C 180,E1 -14008.955,E2 -14008.955} C_VEL
LIN {X 0,Y 340.806,Z 70.033,A -85,B 0,C 180,E1 -14013.02,E2 -14013.02} C_VEL
LIN {X 0,Y 340.733,Z 70.041,A -85,B 0,C 180,E1 -14016.927,E2 -14016.927} C_VEL
LIN {X 0,Y 340.794,Z 70.034,A -85,B 0,C 180,E1 -14020.733,E2 -14020.733} C_VEL
LIN {X 0,Y 340.789,Z 70.032,A -85,B 0,C 180,E1 -14023.218,E2 -14023.218} C_VEL
LIN {X 0,Y 340.847,Z 70.025,A -85,B 0,C 180,E1 -14026.89,E2 -14026.89} C_VEL
LIN {X 0,Y 340.916,Z 70.018,A -85,B 0,C 180,E1 -14030.507,E2 -14030.507} C_VEL
LIN {X 0,Y 341.061,Z 69.998,A -85,B 0,C 180,E1 -14032.898,E2 -14032.898} C_VEL
LIN {X 0,Y 341.169,Z 69.988,A -85,B 0,C 180,E1 -14037.638,E2 -14037.638} C_VEL
LIN {X 0,Y 341.297,Z 69.972,A -85,B 0,C 180,E1 -14040,E2 -14040} C_VEL
LIN {X 0,Y 341.17,Z 69.985,A -85,B 0,C 180,E1 -14042.361,E2 -14042.361} C_VEL
LIN {X 0,Y 341.047,Z 70.001,A -85,B 0,C 180,E1 -14047.102,E2 -14047.102} C_VEL
LIN {X 0,Y 340.85,Z 70.025,A -85,B 0,C 180,E1 -14050.694,E2 -14050.694} C_VEL
LIN {X 0,Y 340.865,Z 70.022,A -85,B 0,C 180,E1 -14054.325,E2 -14054.325} C_VEL
LIN {X 0,Y 340.839,Z 70.026,A -85,B 0,C 180,E1 -14058.466,E2 -14058.466} C_VEL
LIN {X 0,Y 340.719,Z 70.041,A -85,B 0,C 180,E1 -14061.841,E2 -14061.841} C_VEL
LIN {X 0,Y 340.773,Z 70.034,A -85,B 0,C 180,E1 -14065.664,E2 -14065.664} C_VEL
LIN {X 0,Y 340.742,Z 70.039,A -85,B 0,C 180,E1 -14068.319,E2 -14068.319} C_VEL
LIN {X 0,Y 340.705,Z 70.045,A -85,B 0,C 180,E1 -14071.044,E2 -14071.044} C_VEL
LIN {X 0,Y 340.72,Z 70.041,A -85,B 0,C 180,E1 -14075.279,E2 -14075.279} C_VEL
LIN {X 0,Y 340.711,Z 70.047,A -85,B 0,C 180,E1 -14078.386,E2 -14078.386} C_VEL
LIN {X 0,Y 340.7,Z 70.046,A -85,B 0,C 180,E1 -14082.045,E2 -14082.045} C_VEL
LIN {X 0,Y 340.653,Z 70.054,A -85,B 0,C 180,E1 -14086.227,E2 -14086.227} C_VEL
LIN {X 0,Y 340.69,Z 70.047,A -85,B 0,C 180,E1 -14089.753,E2 -14089.753} C_VEL
LIN {X 0,Y 340.707,Z 70.043,A -85,B 0,C 180,E1 -14093.258,E2 -14093.258} C_VEL
LIN {X 0,Y 340.696,Z 70.046,A -85,B 0,C 180,E1 -14096.153,E2 -14096.153} C_VEL
LIN {X 0,Y 340.773,Z 70.172,A -85,B 0,C 180,E1 -14099.329,E2 -14099.329} C_VEL
LIN {X 0,Y 343.486,Z 83.234,A -85,B 0,C 180,E1 -14102.589,E2 -14102.589} C_VEL
LIN {X 0,Y 344.276,Z 88.813,A -85,B 0,C 180,E1 -14103.924,E2 -14103.924} C_VEL
LIN {X 0,Y 342.971,Z 102.935,A -85,B 0,C 180,E1 -14107.086,E2 -14107.086} C_VEL
LIN {X 0,Y 342.654,Z 106.251,A -85,B 0,C 180,E1 -14107.817,E2 -14107.817} C_VEL
LIN {X 0,Y 347.677,Z 146.368,A -85,B 0,C 180,E1 -14108.942,E2 -14108.942} C_VEL
LIN {X 0,Y 346.578,Z 214.833,A -85,B 0,C 180,E1 -14110.375,E2 -14110.375} C_VEL
LIN {X 0,Y 345.968,Z 227.466,A -85,B 0,C 180,E1 -14110.84,E2 -14110.84} C_VEL
LIN {X 0,Y 345.114,Z 239.919,A -85,B 0,C 180,E1 -14111.523,E2 -14111.523} C_VEL
LIN {X 0,Y 344.146,Z 252.463,A -85,B 0,C 180,E1 -14112.469,E2 -14112.469} C_VEL
LIN {X 0,Y 343.084,Z 262.896,A -85,B 0,C 180,E1 -14113.487,E2 -14113.487} C_VEL
LIN {X 0,Y 342.18,Z 273.211,A -85,B 0,C 180,E1 -14114.748,E2 -14114.748} C_VEL
LIN {X 0,Y 341.24,Z 283.44,A -85,B 0,C 180,E1 -14116.299,E2 -14116.299} C_VEL
LIN {X 0,Y 340.484,Z 291.395,A -85,B 0,C 180,E1 -14117.785,E2 -14117.785} C_VEL
LIN {X 0,Y 339.767,Z 299.142,A -85,B 0,C 180,E1 -14119.572,E2 -14119.572} C_VEL
LIN {X 0,Y 339.392,Z 306.292,A -85,B 0,C 180,E1 -14121.665,E2 -14121.665} C_VEL
LIN {X 0,Y 339.16,Z 311.018,A -85,B 0,C 180,E1 -14123.455,E2 -14123.455} C_VEL
LIN {X 0,Y 339.208,Z 314.616,A -85,B 0,C 180,E1 -14125.246,E2 -14125.246} C_VEL
LIN {X 0,Y 339.171,Z 316.439,A -85,B 0,C 180,E1 -14126.436,E2 -14126.436} C_VEL
LIN {X 0,Y 339.221,Z 317.804,A -85,B 0,C 180,E1 -14127.625,E2 -14127.625} C_VEL
LIN {X 0,Y 339.328,Z 318.769,A -85,B 0,C 180,E1 -14128.813,E2 -14128.813} C_VEL
LIN {X 0,Y 339.33,Z 319.332,A -85,B 0,C 180,E1 -14130,E2 -14130} C_VEL
LIN {X 0,Y 339.254,Z 319.474,A -85,B 0,C 180,E1 -14131.187,E2 -14131.187} C_VEL
LIN {X 0,Y 339.113,Z 318.524,A -85,B 0,C 180,E1 -14133.564,E2 -14133.564} C_VEL
LIN {X 0,Y 339.08,Z 316.205,A -85,B 0,C 180,E1 -14135.8,E2 -14135.8} C_VEL
LIN {X 0,Y 339.323,Z 312.987,A -85,B 0,C 180,E1 -14137.737,E2 -14137.737} C_VEL
LIN {X 0,Y 339.697,Z 308.942,A -85,B 0,C 180,E1 -14139.527,E2 -14139.527} C_VEL
LIN {X 0,Y 340.431,Z 302.765,A -85,B 0,C 180,E1 -14141.612,E2 -14141.612} C_VEL
LIN {X 0,Y 341.568,Z 296.066,A -85,B 0,C 180,E1 -14143.384,E2 -14143.384} C_VEL
LIN {X 0,Y 342.787,Z 287.787,A -85,B 0,C 180,E1 -14145.153,E2 -14145.153} C_VEL
LIN {X 0,Y 344.072,Z 279.338,A -85,B 0,C 180,E1 -14146.616,E2 -14146.616} C_VEL
LIN {X 0,Y 345.741,Z 268.937,A -85,B 0,C 180,E1 -14148.058,E2 -14148.058} C_VEL
LIN {X 0,Y 347.238,Z 258.684,A -85,B 0,C 180,E1 -14149.201,E2 -14149.201} C_VEL
LIN {X 0,Y 348.662,Z 247.495,A -85,B 0,C 180,E1 -14150.193,E2 -14150.193} C_VEL
LIN {X 0,Y 350.075,Z 234.941,A -85,B 0,C 180,E1 -14151.029,E2 -14151.029} C_VEL
LIN {X 0,Y 351.189,Z 221.569,A -85,B 0,C 180,E1 -14151.652,E2 -14151.652} C_VEL
LIN {X 0,Y 351.838,Z 208.444,A -85,B 0,C 180,E1 -14152.033,E2 -14152.033} C_VEL
LIN {X 0,Y 353.102,Z 146.973,A -85,B 0,C 180,E1 -14153.318,E2 -14153.318} C_VEL
LIN {X 0,Y 349.617,Z 125.29,A -85,B 0,C 180,E1 -14154.11,E2 -14154.11} C_VEL
LIN {X 0,Y 345.474,Z 105.136,A -85,B 0,C 180,E1 -14154.964,E2 -14154.964} C_VEL
LIN {X 0,Y 346.599,Z 97.02,A -85,B 0,C 180,E1 -14156.85,E2 -14156.85} C_VEL
LIN {X 0,Y 345.945,Z 92.062,A -85,B 0,C 180,E1 -14158.131,E2 -14158.131} C_VEL
LIN {X 0,Y 343.531,Z 81.313,A -85,B 0,C 180,E1 -14161.101,E2 -14161.101} C_VEL
LIN {X 0,Y 341.23,Z 72.13,A -85,B 0,C 180,E1 -14163.786,E2 -14163.786} C_VEL
LIN {X 0,Y 340.726,Z 70.041,A -85,B 0,C 180,E1 -14164.472,E2 -14164.472} C_VEL
LIN {X 0,Y 340.709,Z 70.044,A -85,B 0,C 180,E1 -14168.386,E2 -14168.386} C_VEL
LIN {X 0,Y 340.697,Z 70.045,A -85,B 0,C 180,E1 -14172.045,E2 -14172.045} C_VEL
LIN {X 0,Y 340.664,Z 70.037,A -85,B 0,C 180,E1 -14176.224,E2 -14176.224} C_VEL
LIN {X 0,Y 340.703,Z 70.045,A -85,B 0,C 180,E1 -14178.693,E2 -14178.693} C_VEL
LIN {X 0,Y 340.737,Z 70.037,A -85,B 0,C 180,E1 -14181.773,E2 -14181.773} C_VEL
LIN {X 0,Y 340.721,Z 70.038,A -85,B 0,C 180,E1 -14185.595,E2 -14185.595} C_VEL
LIN {X 0,Y 340.701,Z 70.041,A -85,B 0,C 180,E1 -14188.956,E2 -14188.956} C_VEL
LIN {X 0,Y 340.776,Z 70.033,A -85,B 0,C 180,E1 -14192.474,E2 -14192.474} C_VEL
LIN {X 0,Y 340.753,Z 70.037,A -85,B 0,C 180,E1 -14195.638,E2 -14195.638} C_VEL
LIN {X 0,Y 340.763,Z 70.036,A -85,B 0,C 180,E1 -14199.475,E2 -14199.475} C_VEL
LIN {X 0,Y 340.856,Z 70.017,A -85,B 0,C 180,E1 -14201.984,E2 -14201.984} C_VEL
LIN {X 0,Y 340.866,Z 70.024,A -85,B 0,C 180,E1 -14205.705,E2 -14205.705} C_VEL
LIN {X 0,Y 340.87,Z 70.023,A -85,B 0,C 180,E1 -14209.306,E2 -14209.306} C_VEL
LIN {X 0,Y 341.057,Z 69.992,A -85,B 0,C 180,E1 -14212.898,E2 -14212.898} C_VEL
LIN {X 0,Y 341.165,Z 69.978,A -85,B 0,C 180,E1 -14217.639,E2 -14217.639} C_VEL
LIN {X 0,Y 341.292,Z 69.974,A -85,B 0,C 180,E1 -14220,E2 -14220} C_VEL
LIN {X 0,Y 341.165,Z 69.977,A -85,B 0,C 180,E1 -14222.362,E2 -14222.362} C_VEL
LIN {X 0,Y 341.043,Z 69.998,A -85,B 0,C 180,E1 -14227.103,E2 -14227.103} C_VEL
LIN {X 0,Y 340.846,Z 70.027,A -85,B 0,C 180,E1 -14230.695,E2 -14230.695} C_VEL
LIN {X 0,Y 340.861,Z 70.022,A -85,B 0,C 180,E1 -14234.325,E2 -14234.325} C_VEL
LIN {X 0,Y 340.784,Z 70.029,A -85,B 0,C 180,E1 -14238.441,E2 -14238.441} C_VEL
LIN {X 0,Y 340.716,Z 70.034,A -85,B 0,C 180,E1 -14241.842,E2 -14241.842} C_VEL
LIN {X 0,Y 340.743,Z 70.032,A -85,B 0,C 180,E1 -14245.667,E2 -14245.667} C_VEL
LIN {X 0,Y 340.73,Z 70.036,A -85,B 0,C 180,E1 -14249.672,E2 -14249.672} C_VEL
LIN {X 0,Y 340.691,Z 70.047,A -85,B 0,C 180,E1 -14253.847,E2 -14253.847} C_VEL
LIN {X 0,Y 340.702,Z 70.047,A -85,B 0,C 180,E1 -14256.743,E2 -14256.743} C_VEL
LIN {X 0,Y 340.673,Z 70.044,A -85,B 0,C 180,E1 -14260.245,E2 -14260.245} C_VEL
LIN {X 0,Y 340.651,Z 70.057,A -85,B 0,C 180,E1 -14263.774,E2 -14263.774} C_VEL
LIN {X 0,Y 340.693,Z 70.052,A -85,B 0,C 180,E1 -14267.956,E2 -14267.956} C_VEL
LIN {X 0,Y 340.703,Z 70.136,A -85,B 0,C 180,E1 -14269.57,E2 -14269.57} C_VEL
LIN {X 0,Y 341.59,Z 73.721,A -85,B 0,C 180,E1 -14270.729,E2 -14270.729} C_VEL
LIN {X 0,Y 350.566,Z 92.739,A -85,B 0,C 180,E1 -14272.011,E2 -14272.011} C_VEL
LIN {X 0,Y 354.291,Z 101.773,A -85,B 0,C 180,E1 -14272.544,E2 -14272.544} C_VEL
LIN {X 0,Y 352.379,Z 179.787,A -85,B 0,C 180,E1 -14274.18,E2 -14274.18} C_VEL
LIN {X 0,Y 351.633,Z 193.527,A -85,B 0,C 180,E1 -14274.706,E2 -14274.706} C_VEL
LIN {X 0,Y 350.875,Z 205.499,A -85,B 0,C 180,E1 -14275.401,E2 -14275.401} C_VEL
LIN {X 0,Y 349.748,Z 216.983,A -85,B 0,C 180,E1 -14276.282,E2 -14276.282} C_VEL
LIN {X 0,Y 348.451,Z 227.755,A -85,B 0,C 180,E1 -14277.349,E2 -14277.349} C_VEL
LIN {X 0,Y 346.893,Z 238.779,A -85,B 0,C 180,E1 -14278.725,E2 -14278.725} C_VEL
LIN {X 0,Y 345.504,Z 247.701,A -85,B 0,C 180,E1 -14280.109,E2 -14280.109} C_VEL
LIN {X 0,Y 344.241,Z 255.694,A -85,B 0,C 180,E1 -14281.635,E2 -14281.635} C_VEL
LIN {X 0,Y 342.797,Z 263.618,A -85,B 0,C 180,E1 -14283.519,E2 -14283.519} C_VEL
LIN {X 0,Y 341.796,Z 269.242,A -85,B 0,C 180,E1 -14285.197,E2 -14285.197} C_VEL
LIN {X 0,Y 340.969,Z 273.9,A -85,B 0,C 180,E1 -14286.945,E2 -14286.945} C_VEL
LIN {X 0,Y 340.323,Z 277.745,A -85,B 0,C 180,E1 -14288.841,E2 -14288.841} C_VEL
LIN {X 0,Y 339.778,Z 280.392,A -85,B 0,C 180,E1 -14290.674,E2 -14290.674} C_VEL
LIN {X 0,Y 339.443,Z 281.891,A -85,B 0,C 180,E1 -14292.254,E2 -14292.254} C_VEL
LIN {X 0,Y 339.18,Z 282.777,A -85,B 0,C 180,E1 -14294.374,E2 -14294.374} C_VEL
LIN {X 0,Y 339.131,Z 282.731,A -85,B 0,C 180,E1 -14295.601,E2 -14295.601} C_VEL
LIN {X 0,Y 339.176,Z 282.25,A -85,B 0,C 180,E1 -14296.878,E2 -14296.878} C_VEL
LIN {X 0,Y 339.219,Z 280.084,A -85,B 0,C 180,E1 -14299.254,E2 -14299.254} C_VEL
LIN {X 0,Y 339.489,Z 277.322,A -85,B 0,C 180,E1 -14301.068,E2 -14301.068} C_VEL
LIN {X 0,Y 339.867,Z 273.182,A -85,B 0,C 180,E1 -14303.02,E2 -14303.02} C_VEL
LIN {X 0,Y 340.176,Z 268.638,A -85,B 0,C 180,E1 -14304.666,E2 -14304.666} C_VEL
LIN {X 0,Y 340.755,Z 262.463,A -85,B 0,C 180,E1 -14306.453,E2 -14306.453} C_VEL
LIN {X 0,Y 341.591,Z 254.763,A -85,B 0,C 180,E1 -14308.232,E2 -14308.232} C_VEL
LIN {X 0,Y 342.575,Z 245.106,A -85,B 0,C 180,E1 -14310,E2 -14310} C_VEL
LIN {X 0,Y 343.604,Z 235.131,A -85,B 0,C 180,E1 -14311.465,E2 -14311.465} C_VEL
LIN {X 0,Y 344.619,Z 223.846,A -85,B 0,C 180,E1 -14312.777,E2 -14312.777} C_VEL
LIN {X 0,Y 345.491,Z 212.206,A -85,B 0,C 180,E1 -14313.842,E2 -14313.842} C_VEL
LIN {X 0,Y 346.17,Z 200.612,A -85,B 0,C 180,E1 -14314.658,E2 -14314.658} C_VEL
LIN {X 0,Y 346.658,Z 187.754,A -85,B 0,C 180,E1 -14315.308,E2 -14315.308} C_VEL
LIN {X 0,Y 347.094,Z 173.992,A -85,B 0,C 180,E1 -14315.738,E2 -14315.738} C_VEL
LIN {X 0,Y 348.418,Z 95.94,A -85,B 0,C 180,E1 -14317.344,E2 -14317.344} C_VEL
LIN {X 0,Y 346.794,Z 88.877,A -85,B 0,C 180,E1 -14317.581,E2 -14317.581} C_VEL
LIN {X 0,Y 341.441,Z 72.255,A -85,B 0,C 180,E1 -14318.253,E2 -14318.253} C_VEL
LIN {X 0,Y 340.97,Z 70.013,A -85,B 0,C 180,E1 -14318.916,E2 -14318.916} C_VEL
LIN {X 0,Y 340.849,Z 70.026,A -85,B 0,C 180,E1 -14323.11,E2 -14323.11} C_VEL
LIN {X 0,Y 340.792,Z 70.034,A -85,B 0,C 180,E1 -14326.781,E2 -14326.781} C_VEL
LIN {X 0,Y 340.798,Z 70.031,A -85,B 0,C 180,E1 -14329.266,E2 -14329.266} C_VEL
LIN {X 0,Y 340.708,Z 70.04,A -85,B 0,C 180,E1 -14332.676,E2 -14332.676} C_VEL
LIN {X 0,Y 340.08,Z 70.123,A -85,B 0,C 180,E1 -14333.663,E2 -14333.663} C_VEL
LIN {X 0,Y 337.285,Z 70.477,A -85,B 0,C 180,E1 -14335.27,E2 -14335.27} C_VEL
LIN {X 0,Y 334.879,Z 70.777,A -85,B 0,C 180,E1 -14336.571,E2 -14336.571} C_VEL
LIN {X 0,Y 333.815,Z 70.906,A -85,B 0,C 180,E1 -14337.577,E2 -14337.577} C_VEL
LIN {X 0,Y 333.713,Z 70.916,A -85,B 0,C 180,E1 -14337.918,E2 -14337.918} C_VEL
LIN {X 0,Y 333.695,Z 70.917,A -85,B 0,C 180,E1 -14340.363,E2 -14340.363} C_VEL
LIN {X 0,Y 333.679,Z 70.917,A -85,B 0,C 180,E1 -14344.659,E2 -14344.659} C_VEL
LIN {X 0,Y 333.659,Z 70.926,A -85,B 0,C 180,E1 -14347.651,E2 -14347.651} C_VEL
LIN {X 0,Y 333.651,Z 70.921,A -85,B 0,C 180,E1 -14350.767,E2 -14350.767} C_VEL
LIN {X 0,Y 333.628,Z 70.924,A -85,B 0,C 180,E1 -14354.256,E2 -14354.256} C_VEL
LIN {X 0,Y 333.646,Z 70.924,A -85,B 0,C 180,E1 -14357.618,E2 -14357.618} C_VEL
LIN {X 0,Y 333.656,Z 70.924,A -85,B 0,C 180,E1 -14361.202,E2 -14361.202} C_VEL
LIN {X 0,Y 333.68,Z 70.915,A -85,B 0,C 180,E1 -14363.861,E2 -14363.861} C_VEL
LIN {X 0,Y 333.647,Z 70.922,A -85,B 0,C 180,E1 -14367.413,E2 -14367.413} C_VEL
LIN {X 0,Y 333.693,Z 70.919,A -85,B 0,C 180,E1 -14371.026,E2 -14371.026} C_VEL
LIN {X 0,Y 333.738,Z 70.91,A -85,B 0,C 180,E1 -14373.753,E2 -14373.753} C_VEL
LIN {X 0,Y 333.723,Z 70.912,A -85,B 0,C 180,E1 -14377.914,E2 -14377.914} C_VEL
LIN {X 0,Y 333.797,Z 70.903,A -85,B 0,C 180,E1 -14381.589,E2 -14381.589} C_VEL
LIN {X 0,Y 333.811,Z 70.901,A -85,B 0,C 180,E1 -14385.576,E2 -14385.576} C_VEL
LIN {X 0,Y 333.836,Z 70.898,A -85,B 0,C 180,E1 -14389.078,E2 -14389.078} C_VEL
LIN {X 0,Y 334.008,Z 70.876,A -85,B 0,C 180,E1 -14392.747,E2 -14392.747} C_VEL
LIN {X 0,Y 333.809,Z 70.901,A -85,B 0,C 180,E1 -14395.169,E2 -14395.169} C_VEL
LIN {X 0,Y 334.107,Z 70.867,A -85,B 0,C 180,E1 -14397.589,E2 -14397.589} C_VEL
LIN {X 0,Y 334.248,Z 70.85,A -85,B 0,C 180,E1 -14400,E2 -14400} C_VEL
LIN {X 0,Y 334.107,Z 70.865,A -85,B 0,C 180,E1 -14402.411,E2 -14402.411} C_VEL
LIN {X 0,Y 334.01,Z 70.878,A -85,B 0,C 180,E1 -14406.039,E2 -14406.039} C_VEL
LIN {X 0,Y 333.823,Z 70.903,A -85,B 0,C 180,E1 -14409.696,E2 -14409.696} C_VEL
LIN {X 0,Y 333.799,Z 70.907,A -85,B 0,C 180,E1 -14413.391,E2 -14413.391} C_VEL
LIN {X 0,Y 333.749,Z 70.914,A -85,B 0,C 180,E1 -14417.146,E2 -14417.146} C_VEL
LIN {X 0,Y 333.733,Z 70.912,A -85,B 0,C 180,E1 -14419.69,E2 -14419.69} C_VEL
LIN {X 0,Y 333.671,Z 70.919,A -85,B 0,C 180,E1 -14423.59,E2 -14423.59} C_VEL
LIN {X 0,Y 333.737,Z 70.911,A -85,B 0,C 180,E1 -14426.246,E2 -14426.246} C_VEL
LIN {X 0,Y 333.712,Z 70.916,A -85,B 0,C 180,E1 -14428.972,E2 -14428.972} C_VEL
LIN {X 0,Y 333.645,Z 70.927,A -85,B 0,C 180,E1 -14432.587,E2 -14432.587} C_VEL
LIN {X 0,Y 333.678,Z 70.92,A -85,B 0,C 180,E1 -14436.139,E2 -14436.139} C_VEL
LIN {X 0,Y 333.648,Z 70.921,A -85,B 0,C 180,E1 -14439.192,E2 -14439.192} C_VEL
LIN {X 0,Y 333.634,Z 70.927,A -85,B 0,C 180,E1 -14442.5,E2 -14442.5} C_VEL
LIN {X 0,Y 333.598,Z 70.931,A -85,B 0,C 180,E1 -14445.955,E2 -14445.955} C_VEL
LIN {X 0,Y 333.649,Z 70.922,A -85,B 0,C 180,E1 -14449.315,E2 -14449.315} C_VEL
LIN {X 0,Y 333.667,Z 70.92,A -85,B 0,C 180,E1 -14453.167,E2 -14453.167} C_VEL
LIN {X 0,Y 333.64,Z 70.923,A -85,B 0,C 180,E1 -14456.792,E2 -14456.792} C_VEL
LIN {X 0,Y 333.721,Z 71.045,A -85,B 0,C 180,E1 -14459.036,E2 -14459.036} C_VEL
LIN {X 0,Y 336.415,Z 83.926,A -85,B 0,C 180,E1 -14462.327,E2 -14462.327} C_VEL
LIN {X 0,Y 337.294,Z 89.223,A -85,B 0,C 180,E1 -14463.633,E2 -14463.633} C_VEL
LIN {X 0,Y 336.472,Z 99.364,A -85,B 0,C 180,E1 -14465.964,E2 -14465.964} C_VEL
LIN {X 0,Y 335.754,Z 105.798,A -85,B 0,C 180,E1 -14467.424,E2 -14467.424} C_VEL
LIN {X 0,Y 340.881,Z 146.868,A -85,B 0,C 180,E1 -14468.61,E2 -14468.61} C_VEL
LIN {X 0,Y 339.7,Z 215.323,A -85,B 0,C 180,E1 -14470.079,E2 -14470.079} C_VEL
LIN {X 0,Y 339.096,Z 228.45,A -85,B 0,C 180,E1 -14470.594,E2 -14470.594} C_VEL
LIN {X 0,Y 338.173,Z 240.539,A -85,B 0,C 180,E1 -14471.287,E2 -14471.287} C_VEL
LIN {X 0,Y 337.179,Z 252.785,A -85,B 0,C 180,E1 -14472.251,E2 -14472.251} C_VEL
LIN {X 0,Y 336.094,Z 263.089,A -85,B 0,C 180,E1 -14473.29,E2 -14473.29} C_VEL
LIN {X 0,Y 335.106,Z 273.943,A -85,B 0,C 180,E1 -14474.666,E2 -14474.666} C_VEL
LIN {X 0,Y 334.318,Z 282.555,A -85,B 0,C 180,E1 -14476.01,E2 -14476.01} C_VEL
LIN {X 0,Y 333.501,Z 290.596,A -85,B 0,C 180,E1 -14477.525,E2 -14477.525} C_VEL
LIN {X 0,Y 332.73,Z 298.441,A -85,B 0,C 180,E1 -14479.349,E2 -14479.349} C_VEL
LIN {X 0,Y 332.319,Z 305.651,A -85,B 0,C 180,E1 -14481.486,E2 -14481.486} C_VEL
LIN {X 0,Y 332.093,Z 310.434,A -85,B 0,C 180,E1 -14483.315,E2 -14483.315} C_VEL
LIN {X 0,Y 332.115,Z 314.082,A -85,B 0,C 180,E1 -14485.144,E2 -14485.144} C_VEL
LIN {X 0,Y 332.094,Z 315.948,A -85,B 0,C 180,E1 -14486.36,E2 -14486.36} C_VEL
LIN {X 0,Y 332.126,Z 317.34,A -85,B 0,C 180,E1 -14487.574,E2 -14487.574} C_VEL
LIN {X 0,Y 332.248,Z 318.329,A -85,B 0,C 180,E1 -14488.788,E2 -14488.788} C_VEL
LIN {X 0,Y 332.269,Z 318.915,A -85,B 0,C 180,E1 -14490,E2 -14490} C_VEL
LIN {X 0,Y 332.158,Z 319.094,A -85,B 0,C 180,E1 -14491.212,E2 -14491.212} C_VEL
LIN {X 0,Y 332.034,Z 318.193,A -85,B 0,C 180,E1 -14493.64,E2 -14493.64} C_VEL
LIN {X 0,Y 332.034,Z 315.728,A -85,B 0,C 180,E1 -14496.075,E2 -14496.075} C_VEL
LIN {X 0,Y 332.245,Z 312.749,A -85,B 0,C 180,E1 -14497.902,E2 -14497.902} C_VEL
LIN {X 0,Y 332.661,Z 308.751,A -85,B 0,C 180,E1 -14499.73,E2 -14499.73} C_VEL
LIN {X 0,Y 333.458,Z 302.654,A -85,B 0,C 180,E1 -14501.858,E2 -14501.858} C_VEL
LIN {X 0,Y 334.655,Z 296.016,A -85,B 0,C 180,E1 -14503.665,E2 -14503.665} C_VEL
LIN {X 0,Y 335.934,Z 287.809,A -85,B 0,C 180,E1 -14505.47,E2 -14505.47} C_VEL
LIN {X 0,Y 337.263,Z 279.458,A -85,B 0,C 180,E1 -14506.961,E2 -14506.961} C_VEL
LIN {X 0,Y 339.027,Z 269.219,A -85,B 0,C 180,E1 -14508.429,E2 -14508.429} C_VEL
LIN {X 0,Y 340.554,Z 259.119,A -85,B 0,C 180,E1 -14509.593,E2 -14509.593} C_VEL
LIN {X 0,Y 342.047,Z 248.136,A -85,B 0,C 180,E1 -14510.601,E2 -14510.601} C_VEL
LIN {X 0,Y 343.507,Z 235.988,A -85,B 0,C 180,E1 -14511.451,E2 -14511.451} C_VEL
LIN {X 0,Y 344.67,Z 223.314,A -85,B 0,C 180,E1 -14512.083,E2 -14512.083} C_VEL
LIN {X 0,Y 345.404,Z 210.083,A -85,B 0,C 180,E1 -14512.506,E2 -14512.506} C_VEL
LIN {X 0,Y 346.739,Z 147.443,A -85,B 0,C 180,E1 -14513.848,E2 -14513.848} C_VEL
LIN {X 0,Y 343.334,Z 126.371,A -85,B 0,C 180,E1 -14514.641,E2 -14514.641} C_VEL
LIN {X 0,Y 338.857,Z 104.762,A -85,B 0,C 180,E1 -14515.58,E2 -14515.58} C_VEL
LIN {X 0,Y 339.779,Z 97.97,A -85,B 0,C 180,E1 -14517.2,E2 -14517.2} C_VEL
LIN {X 0,Y 338.24,Z 89.605,A -85,B 0,C 180,E1 -14519.482,E2 -14519.482} C_VEL
LIN {X 0,Y 335.356,Z 77.351,A -85,B 0,C 180,E1 -14523.042,E2 -14523.042} C_VEL
LIN {X 0,Y 333.663,Z 70.918,A -85,B 0,C 180,E1 -14525.03,E2 -14525.03} C_VEL
LIN {X 0,Y 333.652,Z 70.923,A -85,B 0,C 180,E1 -14528.798,E2 -14528.798} C_VEL
LIN {X 0,Y 333.631,Z 70.926,A -85,B 0,C 180,E1 -14532.5,E2 -14532.5} C_VEL
LIN {X 0,Y 333.606,Z 70.914,A -85,B 0,C 180,E1 -14535.957,E2 -14535.957} C_VEL
LIN {X 0,Y 333.654,Z 70.92,A -85,B 0,C 180,E1 -14539.313,E2 -14539.313} C_VEL
LIN {X 0,Y 333.654,Z 70.917,A -85,B 0,C 180,E1 -14542.349,E2 -14542.349} C_VEL
LIN {X 0,Y 333.672,Z 70.916,A -85,B 0,C 180,E1 -14545.341,E2 -14545.341} C_VEL
LIN {X 0,Y 333.695,Z 70.913,A -85,B 0,C 180,E1 -14549.638,E2 -14549.638} C_VEL
LIN {X 0,Y 333.741,Z 70.91,A -85,B 0,C 180,E1 -14552.401,E2 -14552.401} C_VEL
LIN {X 0,Y 333.725,Z 70.916,A -85,B 0,C 180,E1 -14555.091,E2 -14555.091} C_VEL
LIN {X 0,Y 333.691,Z 70.919,A -85,B 0,C 180,E1 -14559.02,E2 -14559.02} C_VEL
LIN {X 0,Y 333.793,Z 70.899,A -85,B 0,C 180,E1 -14561.59,E2 -14561.59} C_VEL
LIN {X 0,Y 333.805,Z 70.903,A -85,B 0,C 180,E1 -14565.577,E2 -14565.577} C_VEL
LIN {X 0,Y 333.832,Z 70.9,A -85,B 0,C 180,E1 -14569.078,E2 -14569.078} C_VEL
LIN {X 0,Y 334.01,Z 70.869,A -85,B 0,C 180,E1 -14572.747,E2 -14572.747} C_VEL
LIN {X 0,Y 333.806,Z 70.904,A -85,B 0,C 180,E1 -14575.169,E2 -14575.169} C_VEL
LIN {X 0,Y 334.102,Z 70.857,A -85,B 0,C 180,E1 -14577.589,E2 -14577.589} C_VEL
LIN {X 0,Y 334.243,Z 70.852,A -85,B 0,C 180,E1 -14580,E2 -14580} C_VEL
LIN {X 0,Y 334.102,Z 70.856,A -85,B 0,C 180,E1 -14582.411,E2 -14582.411} C_VEL
LIN {X 0,Y 333.979,Z 70.876,A -85,B 0,C 180,E1 -14586.606,E2 -14586.606} C_VEL
LIN {X 0,Y 333.819,Z 70.903,A -85,B 0,C 180,E1 -14589.697,E2 -14589.697} C_VEL
LIN {X 0,Y 333.795,Z 70.898,A -85,B 0,C 180,E1 -14593.392,E2 -14593.392} C_VEL
LIN {X 0,Y 333.717,Z 70.908,A -85,B 0,C 180,E1 -14597.148,E2 -14597.148} C_VEL
LIN {X 0,Y 333.687,Z 70.919,A -85,B 0,C 180,E1 -14599.694,E2 -14599.694} C_VEL
LIN {X 0,Y 333.667,Z 70.921,A -85,B 0,C 180,E1 -14603.591,E2 -14603.591} C_VEL
LIN {X 0,Y 333.674,Z 70.914,A -85,B 0,C 180,E1 -14606.252,E2 -14606.252} C_VEL
LIN {X 0,Y 333.658,Z 70.922,A -85,B 0,C 180,E1 -14610.367,E2 -14610.367} C_VEL
LIN {X 0,Y 333.636,Z 70.925,A -85,B 0,C 180,E1 -14613.209,E2 -14613.209} C_VEL
LIN {X 0,Y 333.674,Z 70.921,A -85,B 0,C 180,E1 -14616.14,E2 -14616.14} C_VEL
LIN {X 0,Y 333.631,Z 70.93,A -85,B 0,C 180,E1 -14619.195,E2 -14619.195} C_VEL
LIN {X 0,Y 333.63,Z 70.928,A -85,B 0,C 180,E1 -14622.5,E2 -14622.5} C_VEL
LIN {X 0,Y 333.595,Z 70.931,A -85,B 0,C 180,E1 -14625.956,E2 -14625.956} C_VEL
LIN {X 0,Y 333.659,Z 71.021,A -85,B 0,C 180,E1 -14628.986,E2 -14628.986} C_VEL
LIN {X 0,Y 334.333,Z 73.905,A -85,B 0,C 180,E1 -14629.992,E2 -14629.992} C_VEL
LIN {X 0,Y 343.753,Z 93.486,A -85,B 0,C 180,E1 -14631.408,E2 -14631.408} C_VEL
LIN {X 0,Y 347.964,Z 103.563,A -85,B 0,C 180,E1 -14632.029,E2 -14632.029} C_VEL
LIN {X 0,Y 346.006,Z 180.512,A -85,B 0,C 180,E1 -14633.676,E2 -14633.676} C_VEL
LIN {X 0,Y 345.23,Z 194.331,A -85,B 0,C 180,E1 -14634.221,E2 -14634.221} C_VEL
LIN {X 0,Y 344.491,Z 205.339,A -85,B 0,C 180,E1 -14634.87,E2 -14634.87} C_VEL
LIN {X 0,Y 343.359,Z 216.723,A -85,B 0,C 180,E1 -14635.745,E2 -14635.745} C_VEL
LIN {X 0,Y 341.993,Z 227.637,A -85,B 0,C 180,E1 -14636.829,E2 -14636.829} C_VEL
LIN {X 0,Y 340.336,Z 238.96,A -85,B 0,C 180,E1 -14638.258,E2 -14638.258} C_VEL
LIN {X 0,Y 338.735,Z 248.645,A -85,B 0,C 180,E1 -14639.793,E2 -14639.793} C_VEL
LIN {X 0,Y 337.403,Z 256.634,A -85,B 0,C 180,E1 -14641.375,E2 -14641.375} C_VEL
LIN {X 0,Y 335.907,Z 264.355,A -85,B 0,C 180,E1 -14643.268,E2 -14643.268} C_VEL
LIN {X 0,Y 334.758,Z 270.477,A -85,B 0,C 180,E1 -14645.173,E2 -14645.173} C_VEL
LIN {X 0,Y 333.868,Z 275.234,A -85,B 0,C 180,E1 -14647.082,E2 -14647.082} C_VEL
LIN {X 0,Y 333.193,Z 278.785,A -85,B 0,C 180,E1 -14648.988,E2 -14648.988} C_VEL
LIN {X 0,Y 332.801,Z 280.522,A -85,B 0,C 180,E1 -14650.253,E2 -14650.253} C_VEL
LIN {X 0,Y 332.397,Z 282.271,A -85,B 0,C 180,E1 -14652.076,E2 -14652.076} C_VEL
LIN {X 0,Y 332.115,Z 283.141,A -85,B 0,C 180,E1 -14654.033,E2 -14654.033} C_VEL
LIN {X 0,Y 332.056,Z 283.152,A -85,B 0,C 180,E1 -14655.287,E2 -14655.287} C_VEL
LIN {X 0,Y 332.096,Z 282.656,A -85,B 0,C 180,E1 -14656.778,E2 -14656.778} C_VEL
LIN {X 0,Y 332.122,Z 280.73,A -85,B 0,C 180,E1 -14659.022,E2 -14659.022} C_VEL
LIN {X 0,Y 332.379,Z 278.086,A -85,B 0,C 180,E1 -14660.876,E2 -14660.876} C_VEL
LIN {X 0,Y 332.774,Z 273.677,A -85,B 0,C 180,E1 -14663.037,E2 -14663.037} C_VEL
LIN {X 0,Y 333.259,Z 267.82,A -85,B 0,C 180,E1 -14665.162,E2 -14665.162} C_VEL
LIN {X 0,Y 333.88,Z 261.315,A -85,B 0,C 180,E1 -14666.984,E2 -14666.984} C_VEL
LIN {X 0,Y 334.811,Z 253.209,A -85,B 0,C 180,E1 -14668.798,E2 -14668.798} C_VEL
LIN {X 0,Y 335.679,Z 244.951,A -85,B 0,C 180,E1 -14670.3,E2 -14670.3} C_VEL
LIN {X 0,Y 336.708,Z 234.84,A -85,B 0,C 180,E1 -14671.795,E2 -14671.795} C_VEL
LIN {X 0,Y 337.786,Z 223.458,A -85,B 0,C 180,E1 -14673.123,E2 -14673.123} C_VEL
LIN {X 0,Y 338.622,Z 212.525,A -85,B 0,C 180,E1 -14674.135,E2 -14674.135} C_VEL
LIN {X 0,Y 339.345,Z 200.756,A -85,B 0,C 180,E1 -14674.976,E2 -14674.976} C_VEL
LIN {X 0,Y 339.845,Z 187.785,A -85,B 0,C 180,E1 -14675.638,E2 -14675.638} C_VEL
LIN {X 0,Y 340.28,Z 173.851,A -85,B 0,C 180,E1 -14676.076,E2 -14676.076} C_VEL
LIN {X 0,Y 341.579,Z 96.4,A -85,B 0,C 180,E1 -14677.7,E2 -14677.7} C_VEL
LIN {X 0,Y 339.54,Z 88.57,A -85,B 0,C 180,E1 -14677.985,E2 -14677.985} C_VEL
LIN {X 0,Y 334.285,Z 72.658,A -85,B 0,C 180,E1 -14678.648,E2 -14678.648} C_VEL
LIN {X 0,Y 333.903,Z 70.891,A -85,B 0,C 180,E1 -14679.236,E2 -14679.236} C_VEL
LIN {X 0,Y 333.802,Z 70.903,A -85,B 0,C 180,E1 -14683.392,E2 -14683.392} C_VEL
LIN {X 0,Y 333.752,Z 70.909,A -85,B 0,C 180,E1 -14687.146,E2 -14687.146} C_VEL
LIN {X 0,Y 333.74,Z 70.911,A -85,B 0,C 180,E1 -14689.691,E2 -14689.691} C_VEL
LIN {X 0,Y 333.675,Z 70.919,A -85,B 0,C 180,E1 -14693.59,E2 -14693.59} C_VEL
LIN {X 0,Y 333.739,Z 70.913,A -85,B 0,C 180,E1 -14696.246,E2 -14696.246} C_VEL
LIN {X 0,Y 333.713,Z 70.916,A -85,B 0,C 180,E1 -14697.918,E2 -14697.918} C_VEL
LIN {X 0,Y 333.005,Z 71.002,A -85,B 0,C 180,E1 -14698.924,E2 -14698.924} C_VEL
LIN {X 0,Y 330.144,Z 71.358,A -85,B 0,C 180,E1 -14700.562,E2 -14700.562} C_VEL
LIN {X 0,Y 327.739,Z 71.662,A -85,B 0,C 180,E1 -14701.889,E2 -14701.889} C_VEL
LIN {X 0,Y 326.699,Z 71.786,A -85,B 0,C 180,E1 -14702.915,E2 -14702.915} C_VEL
LIN {X 0,Y 326.608,Z 71.797,A -85,B 0,C 180,E1 -14703.263,E2 -14703.263} C_VEL
LIN {X 0,Y 326.637,Z 71.796,A -85,B 0,C 180,E1 -14707.046,E2 -14707.046} C_VEL
LIN {X 0,Y 326.596,Z 71.8,A -85,B 0,C 180,E1 -14710.209,E2 -14710.209} C_VEL
LIN {X 0,Y 326.579,Z 71.806,A -85,B 0,C 180,E1 -14713.523,E2 -14713.523} C_VEL
LIN {X 0,Y 326.586,Z 71.804,A -85,B 0,C 180,E1 -14717.027,E2 -14717.027} C_VEL
LIN {X 0,Y 326.615,Z 71.799,A -85,B 0,C 180,E1 -14720.773,E2 -14720.773} C_VEL
LIN {X 0,Y 326.616,Z 71.794,A -85,B 0,C 180,E1 -14724.48,E2 -14724.48} C_VEL
LIN {X 0,Y 326.611,Z 71.798,A -85,B 0,C 180,E1 -14727.455,E2 -14727.455} C_VEL
LIN {X 0,Y 326.651,Z 71.794,A -85,B 0,C 180,E1 -14730.339,E2 -14730.339} C_VEL
LIN {X 0,Y 326.693,Z 71.791,A -85,B 0,C 180,E1 -14734.516,E2 -14734.516} C_VEL
LIN {X 0,Y 326.652,Z 71.798,A -85,B 0,C 180,E1 -14738.545,E2 -14738.545} C_VEL
LIN {X 0,Y 326.748,Z 71.781,A -85,B 0,C 180,E1 -14741.177,E2 -14741.177} C_VEL
LIN {X 0,Y 326.766,Z 71.778,A -85,B 0,C 180,E1 -14745.433,E2 -14745.433} C_VEL
LIN {X 0,Y 326.773,Z 71.778,A -85,B 0,C 180,E1 -14748.839,E2 -14748.839} C_VEL
LIN {X 0,Y 326.961,Z 71.755,A -85,B 0,C 180,E1 -14752.59,E2 -14752.59} C_VEL
LIN {X 0,Y 326.776,Z 71.777,A -85,B 0,C 180,E1 -14755.065,E2 -14755.065} C_VEL
LIN {X 0,Y 327.047,Z 71.746,A -85,B 0,C 180,E1 -14757.536,E2 -14757.536} C_VEL
LIN {X 0,Y 327.199,Z 71.727,A -85,B 0,C 180,E1 -14760,E2 -14760} C_VEL
LIN {X 0,Y 327.047,Z 71.744,A -85,B 0,C 180,E1 -14762.463,E2 -14762.463} C_VEL
LIN {X 0,Y 326.984,Z 71.752,A -85,B 0,C 180,E1 -14766.169,E2 -14766.169} C_VEL
LIN {X 0,Y 326.785,Z 71.778,A -85,B 0,C 180,E1 -14769.907,E2 -14769.907} C_VEL
LIN {X 0,Y 326.761,Z 71.781,A -85,B 0,C 180,E1 -14773.685,E2 -14773.685} C_VEL
LIN {X 0,Y 326.701,Z 71.789,A -85,B 0,C 180,E1 -14777.528,E2 -14777.528} C_VEL
LIN {X 0,Y 326.66,Z 71.792,A -85,B 0,C 180,E1 -14780.135,E2 -14780.135} C_VEL
LIN {X 0,Y 326.65,Z 71.793,A -85,B 0,C 180,E1 -14784.129,E2 -14784.129} C_VEL
LIN {X 0,Y 326.686,Z 71.794,A -85,B 0,C 180,E1 -14786.857,E2 -14786.857} C_VEL
LIN {X 0,Y 326.641,Z 71.798,A -85,B 0,C 180,E1 -14790.611,E2 -14790.611} C_VEL
LIN {X 0,Y 326.608,Z 71.799,A -85,B 0,C 180,E1 -14794.019,E2 -14794.019} C_VEL
LIN {X 0,Y 326.629,Z 71.796,A -85,B 0,C 180,E1 -14797.238,E2 -14797.238} C_VEL
LIN {X 0,Y 326.579,Z 71.802,A -85,B 0,C 180,E1 -14801.131,E2 -14801.131} C_VEL
LIN {X 0,Y 326.529,Z 71.809,A -85,B 0,C 180,E1 -14804.743,E2 -14804.743} C_VEL
LIN {X 0,Y 326.578,Z 71.808,A -85,B 0,C 180,E1 -14808.154,E2 -14808.154} C_VEL
LIN {X 0,Y 326.625,Z 71.798,A -85,B 0,C 180,E1 -14811.391,E2 -14811.391} C_VEL
LIN {X 0,Y 326.621,Z 71.797,A -85,B 0,C 180,E1 -14814.851,E2 -14814.851} C_VEL
LIN {X 0,Y 326.644,Z 71.921,A -85,B 0,C 180,E1 -14818.73,E2 -14818.73} C_VEL
LIN {X 0,Y 329.296,Z 84.382,A -85,B 0,C 180,E1 -14821.995,E2 -14821.995} C_VEL
LIN {X 0,Y 330.291,Z 90.171,A -85,B 0,C 180,E1 -14823.458,E2 -14823.458} C_VEL
LIN {X 0,Y 329.492,Z 99.958,A -85,B 0,C 180,E1 -14825.757,E2 -14825.757} C_VEL
LIN {X 0,Y 328.857,Z 105.444,A -85,B 0,C 180,E1 -14827.03,E2 -14827.03} C_VEL
LIN {X 0,Y 334.055,Z 146.882,A -85,B 0,C 180,E1 -14828.254,E2 -14828.254} C_VEL
LIN {X 0,Y 332.899,Z 214.635,A -85,B 0,C 180,E1 -14829.735,E2 -14829.735} C_VEL
LIN {X 0,Y 332.22,Z 227.85,A -85,B 0,C 180,E1 -14830.256,E2 -14830.256} C_VEL
LIN {X 0,Y 331.347,Z 240.019,A -85,B 0,C 180,E1 -14830.967,E2 -14830.967} C_VEL
LIN {X 0,Y 330.309,Z 251.488,A -85,B 0,C 180,E1 -14831.869,E2 -14831.869} C_VEL
LIN {X 0,Y 329.222,Z 261.971,A -85,B 0,C 180,E1 -14832.93,E2 -14832.93} C_VEL
LIN {X 0,Y 328.217,Z 272.86,A -85,B 0,C 180,E1 -14834.322,E2 -14834.322} C_VEL
LIN {X 0,Y 327.394,Z 281.669,A -85,B 0,C 180,E1 -14835.708,E2 -14835.708} C_VEL
LIN {X 0,Y 326.529,Z 289.792,A -85,B 0,C 180,E1 -14837.254,E2 -14837.254} C_VEL
LIN {X 0,Y 325.688,Z 297.738,A -85,B 0,C 180,E1 -14839.116,E2 -14839.116} C_VEL
LIN {X 0,Y 325.34,Z 303.14,A -85,B 0,C 180,E1 -14840.676,E2 -14840.676} C_VEL
LIN {X 0,Y 325.077,Z 308.394,A -85,B 0,C 180,E1 -14842.546,E2 -14842.546} C_VEL
LIN {X 0,Y 324.962,Z 311.992,A -85,B 0,C 180,E1 -14844.183,E2 -14844.183} C_VEL
LIN {X 0,Y 325.019,Z 315.447,A -85,B 0,C 180,E1 -14846.28,E2 -14846.28} C_VEL
LIN {X 0,Y 325.032,Z 316.876,A -85,B 0,C 180,E1 -14847.521,E2 -14847.521} C_VEL
LIN {X 0,Y 325.152,Z 317.888,A -85,B 0,C 180,E1 -14848.761,E2 -14848.761} C_VEL
LIN {X 0,Y 325.191,Z 318.497,A -85,B 0,C 180,E1 -14850,E2 -14850} C_VEL
LIN {X 0,Y 325.062,Z 318.704,A -85,B 0,C 180,E1 -14851.238,E2 -14851.238} C_VEL
LIN {X 0,Y 324.952,Z 318.483,A -85,B 0,C 180,E1 -14852.479,E2 -14852.479} C_VEL
LIN {X 0,Y 324.956,Z 317.862,A -85,B 0,C 180,E1 -14853.72,E2 -14853.72} C_VEL
LIN {X 0,Y 324.953,Z 315.445,A -85,B 0,C 180,E1 -14856.208,E2 -14856.208} C_VEL
LIN {X 0,Y 325.183,Z 312.508,A -85,B 0,C 180,E1 -14858.075,E2 -14858.075} C_VEL
LIN {X 0,Y 325.615,Z 308.561,A -85,B 0,C 180,E1 -14859.943,E2 -14859.943} C_VEL
LIN {X 0,Y 326.333,Z 303.509,A -85,B 0,C 180,E1 -14861.805,E2 -14861.805} C_VEL
LIN {X 0,Y 327.525,Z 297.202,A -85,B 0,C 180,E1 -14863.652,E2 -14863.652} C_VEL
LIN {X 0,Y 328.795,Z 289.496,A -85,B 0,C 180,E1 -14865.465,E2 -14865.465} C_VEL
LIN {X 0,Y 330.137,Z 281.553,A -85,B 0,C 180,E1 -14866.988,E2 -14866.988} C_VEL
LIN {X 0,Y 331.933,Z 271.68,A -85,B 0,C 180,E1 -14868.517,E2 -14868.517} C_VEL
LIN {X 0,Y 333.611,Z 260.946,A -85,B 0,C 180,E1 -14869.858,E2 -14869.858} C_VEL
LIN {X 0,Y 335.238,Z 250.531,A -85,B 0,C 180,E1 -14870.878,E2 -14870.878} C_VEL
LIN {X 0,Y 336.82,Z 238.047,A -85,B 0,C 180,E1 -14871.818,E2 -14871.818} C_VEL
LIN {X 0,Y 338.161,Z 224.911,A -85,B 0,C 180,E1 -14872.531,E2 -14872.531} C_VEL
LIN {X 0,Y 339.015,Z 211.699,A -85,B 0,C 180,E1 -14872.994,E2 -14872.994} C_VEL
LIN {X 0,Y 340.533,Z 149.182,A -85,B 0,C 180,E1 -14874.355,E2 -14874.355} C_VEL
LIN {X 0,Y 337.321,Z 128.711,A -85,B 0,C 180,E1 -14875.143,E2 -14875.143} C_VEL
LIN {X 0,Y 332.28,Z 104.436,A -85,B 0,C 180,E1 -14876.229,E2 -14876.229} C_VEL
LIN {X 0,Y 332.939,Z 99.001,A -85,B 0,C 180,E1 -14877.554,E2 -14877.554} C_VEL
LIN {X 0,Y 330.928,Z 89.126,A -85,B 0,C 180,E1 -14880.339,E2 -14880.339} C_VEL
LIN {X 0,Y 328.475,Z 78.8,A -85,B 0,C 180,E1 -14883.443,E2 -14883.443} C_VEL
LIN {X 0,Y 326.631,Z 71.796,A -85,B 0,C 180,E1 -14885.706,E2 -14885.706} C_VEL
LIN {X 0,Y 326.61,Z 71.802,A -85,B 0,C 180,E1 -14889.227,E2 -14889.227} C_VEL
LIN {X 0,Y 326.574,Z 71.806,A -85,B 0,C 180,E1 -14892.972,E2 -14892.972} C_VEL
LIN {X 0,Y 326.597,Z 71.797,A -85,B 0,C 180,E1 -14897.023,E2 -14897.023} C_VEL
LIN {X 0,Y 326.632,Z 71.798,A -85,B 0,C 180,E1 -14900.767,E2 -14900.767} C_VEL
LIN {X 0,Y 326.611,Z 71.8,A -85,B 0,C 180,E1 -14904.48,E2 -14904.48} C_VEL
LIN {X 0,Y 326.607,Z 71.802,A -85,B 0,C 180,E1 -14907.456,E2 -14907.456} C_VEL
LIN {X 0,Y 326.658,Z 71.791,A -85,B 0,C 180,E1 -14910.341,E2 -14910.341} C_VEL
LIN {X 0,Y 326.687,Z 71.788,A -85,B 0,C 180,E1 -14914.516,E2 -14914.516} C_VEL
LIN {X 0,Y 326.65,Z 71.789,A -85,B 0,C 180,E1 -14918.546,E2 -14918.546} C_VEL
LIN {X 0,Y 326.742,Z 71.778,A -85,B 0,C 180,E1 -14921.178,E2 -14921.178} C_VEL
LIN {X 0,Y 326.76,Z 71.78,A -85,B 0,C 180,E1 -14925.433,E2 -14925.433} C_VEL
LIN {X 0,Y 326.768,Z 71.78,A -85,B 0,C 180,E1 -14928.839,E2 -14928.839} C_VEL
LIN {X 0,Y 326.963,Z 71.746,A -85,B 0,C 180,E1 -14932.59,E2 -14932.59} C_VEL
LIN {X 0,Y 326.773,Z 71.78,A -85,B 0,C 180,E1 -14935.065,E2 -14935.065} C_VEL
LIN {X 0,Y 327.043,Z 71.736,A -85,B 0,C 180,E1 -14937.537,E2 -14937.537} C_VEL
LIN {X 0,Y 327.194,Z 71.73,A -85,B 0,C 180,E1 -14940,E2 -14940} C_VEL
LIN {X 0,Y 327.043,Z 71.735,A -85,B 0,C 180,E1 -14942.464,E2 -14942.464} C_VEL
LIN {X 0,Y 326.948,Z 71.752,A -85,B 0,C 180,E1 -14946.595,E2 -14946.595} C_VEL
LIN {X 0,Y 326.781,Z 71.78,A -85,B 0,C 180,E1 -14949.908,E2 -14949.908} C_VEL
LIN {X 0,Y 326.757,Z 71.776,A -85,B 0,C 180,E1 -14953.686,E2 -14953.686} C_VEL
LIN {X 0,Y 326.662,Z 71.785,A -85,B 0,C 180,E1 -14957.53,E2 -14957.53} C_VEL
LIN {X 0,Y 326.632,Z 71.798,A -85,B 0,C 180,E1 -14960.137,E2 -14960.137} C_VEL
LIN {X 0,Y 326.642,Z 71.797,A -85,B 0,C 180,E1 -14964.13,E2 -14964.13} C_VEL
LIN {X 0,Y 326.626,Z 71.799,A -85,B 0,C 180,E1 -14968.254,E2 -14968.254} C_VEL
LIN {X 0,Y 326.574,Z 71.805,A -85,B 0,C 180,E1 -14971.098,E2 -14971.098} C_VEL
LIN {X 0,Y 326.606,Z 71.803,A -85,B 0,C 180,E1 -14974.02,E2 -14974.02} C_VEL
LIN {X 0,Y 326.622,Z 71.8,A -85,B 0,C 180,E1 -14977.238,E2 -14977.238} C_VEL
LIN {X 0,Y 326.573,Z 71.795,A -85,B 0,C 180,E1 -14981.131,E2 -14981.131} C_VEL
LIN {X 0,Y 326.526,Z 71.807,A -85,B 0,C 180,E1 -14984.743,E2 -14984.743} C_VEL
LIN {X 0,Y 326.633,Z 71.999,A -85,B 0,C 180,E1 -14988.412,E2 -14988.412} C_VEL
LIN {X 0,Y 327.2,Z 74.405,A -85,B 0,C 180,E1 -14989.272,E2 -14989.272} C_VEL
LIN {X 0,Y 336.555,Z 93.349,A -85,B 0,C 180,E1 -14990.71,E2 -14990.71} C_VEL
LIN {X 0,Y 341.728,Z 105.454,A -85,B 0,C 180,E1 -14991.502,E2 -14991.502} C_VEL
LIN {X 0,Y 339.707,Z 180.588,A -85,B 0,C 180,E1 -14993.133,E2 -14993.133} C_VEL
LIN {X 0,Y 338.914,Z 194.023,A -85,B 0,C 180,E1 -14993.661,E2 -14993.661} C_VEL
LIN {X 0,Y 338.032,Z 206.387,A -85,B 0,C 180,E1 -14994.399,E2 -14994.399} C_VEL
LIN {X 0,Y 336.771,Z 218.182,A -85,B 0,C 180,E1 -14995.343,E2 -14995.343} C_VEL
LIN {X 0,Y 335.185,Z 230.227,A -85,B 0,C 180,E1 -14996.606,E2 -14996.606} C_VEL
LIN {X 0,Y 333.593,Z 240.298,A -85,B 0,C 180,E1 -14997.936,E2 -14997.936} C_VEL
LIN {X 0,Y 331.966,Z 249.566,A -85,B 0,C 180,E1 -14999.463,E2 -14999.463} C_VEL
LIN {X 0,Y 330.572,Z 257.462,A -85,B 0,C 180,E1 -15001.075,E2 -15001.075} C_VEL
LIN {X 0,Y 329.034,Z 265.105,A -85,B 0,C 180,E1 -15003.007,E2 -15003.007} C_VEL
LIN {X 0,Y 327.974,Z 270.224,A -85,B 0,C 180,E1 -15004.624,E2 -15004.624} C_VEL
LIN {X 0,Y 327.019,Z 275.122,A -85,B 0,C 180,E1 -15006.573,E2 -15006.573} C_VEL
LIN {X 0,Y 326.285,Z 278.805,A -85,B 0,C 180,E1 -15008.521,E2 -15008.521} C_VEL
LIN {X 0,Y 325.848,Z 280.656,A -85,B 0,C 180,E1 -15009.813,E2 -15009.813} C_VEL
LIN {X 0,Y 325.34,Z 282.657,A -85,B 0,C 180,E1 -15011.897,E2 -15011.897} C_VEL
LIN {X 0,Y 325.063,Z 283.498,A -85,B 0,C 180,E1 -15013.677,E2 -15013.677} C_VEL
LIN {X 0,Y 324.98,Z 283.572,A -85,B 0,C 180,E1 -15014.959,E2 -15014.959} C_VEL
LIN {X 0,Y 325.003,Z 283.056,A -85,B 0,C 180,E1 -15016.683,E2 -15016.683} C_VEL
LIN {X 0,Y 325.035,Z 281.375,A -85,B 0,C 180,E1 -15018.779,E2 -15018.779} C_VEL
LIN {X 0,Y 325.239,Z 278.852,A -85,B 0,C 180,E1 -15020.674,E2 -15020.674} C_VEL
LIN {X 0,Y 325.692,Z 274.208,A -85,B 0,C 180,E1 -15023.039,E2 -15023.039} C_VEL
LIN {X 0,Y 326.126,Z 268.857,A -85,B 0,C 180,E1 -15025.055,E2 -15025.055} C_VEL
LIN {X 0,Y 326.784,Z 262.545,A -85,B 0,C 180,E1 -15026.918,E2 -15026.918} C_VEL
LIN {X 0,Y 327.677,Z 254.631,A -85,B 0,C 180,E1 -15028.771,E2 -15028.771} C_VEL
LIN {X 0,Y 328.558,Z 246.573,A -85,B 0,C 180,E1 -15030.307,E2 -15030.307} C_VEL
LIN {X 0,Y 329.652,Z 236.734,A -85,B 0,C 180,E1 -15031.833,E2 -15031.833} C_VEL
LIN {X 0,Y 330.614,Z 227.076,A -85,B 0,C 180,E1 -15033.047,E2 -15033.047} C_VEL
LIN {X 0,Y 331.562,Z 215.644,A -85,B 0,C 180,E1 -15034.195,E2 -15034.195} C_VEL
LIN {X 0,Y 332.363,Z 203.134,A -85,B 0,C 180,E1 -15035.156,E2 -15035.156} C_VEL
LIN {X 0,Y 332.959,Z 190.385,A -85,B 0,C 180,E1 -15035.869,E2 -15035.869} C_VEL
LIN {X 0,Y 333.388,Z 177.312,A -85,B 0,C 180,E1 -15036.332,E2 -15036.332} C_VEL
LIN {X 0,Y 334.818,Z 97.324,A -85,B 0,C 180,E1 -15038.055,E2 -15038.055} C_VEL
LIN {X 0,Y 330.124,Z 81.619,A -85,B 0,C 180,E1 -15038.68,E2 -15038.68} C_VEL
LIN {X 0,Y 327.117,Z 72.988,A -85,B 0,C 180,E1 -15039.082,E2 -15039.082} C_VEL
LIN {X 0,Y 326.858,Z 71.769,A -85,B 0,C 180,E1 -15039.515,E2 -15039.515} C_VEL
LIN {X 0,Y 326.764,Z 71.781,A -85,B 0,C 180,E1 -15043.686,E2 -15043.686} C_VEL
LIN {X 0,Y 326.705,Z 71.787,A -85,B 0,C 180,E1 -15047.528,E2 -15047.528} C_VEL
LIN {X 0,Y 326.665,Z 71.796,A -85,B 0,C 180,E1 -15050.135,E2 -15050.135} C_VEL
LIN {X 0,Y 326.654,Z 71.798,A -85,B 0,C 180,E1 -15054.129,E2 -15054.129} C_VEL
LIN {X 0,Y 326.687,Z 71.788,A -85,B 0,C 180,E1 -15056.858,E2 -15056.858} C_VEL
LIN {X 0,Y 326.639,Z 71.795,A -85,B 0,C 180,E1 -15060.61,E2 -15060.61} C_VEL
LIN {X 0,Y 326.608,Z 71.797,A -85,B 0,C 180,E1 -15063.263,E2 -15063.263} C_VEL
LIN {X 0,Y 325.927,Z 71.885,A -85,B 0,C 180,E1 -15064.292,E2 -15064.292} C_VEL
LIN {X 0,Y 323.076,Z 72.241,A -85,B 0,C 180,E1 -15065.967,E2 -15065.967} C_VEL
LIN {X 0,Y 320.665,Z 72.541,A -85,B 0,C 180,E1 -15067.324,E2 -15067.324} C_VEL
LIN {X 0,Y 319.624,Z 72.669,A -85,B 0,C 180,E1 -15068.374,E2 -15068.374} C_VEL
LIN {X 0,Y 319.535,Z 72.678,A -85,B 0,C 180,E1 -15068.73,E2 -15068.73} C_VEL
LIN {X 0,Y 319.564,Z 72.677,A -85,B 0,C 180,E1 -15072.982,E2 -15072.982} C_VEL
LIN {X 0,Y 319.565,Z 72.678,A -85,B 0,C 180,E1 -15077.018,E2 -15077.018} C_VEL
LIN {X 0,Y 319.55,Z 72.677,A -85,B 0,C 180,E1 -15080.371,E2 -15080.371} C_VEL
LIN {X 0,Y 319.583,Z 72.668,A -85,B 0,C 180,E1 -15084.457,E2 -15084.457} C_VEL
LIN {X 0,Y 319.534,Z 72.678,A -85,B 0,C 180,E1 -15088.138,E2 -15088.138} C_VEL
LIN {X 0,Y 319.614,Z 72.67,A -85,B 0,C 180,E1 -15091.59,E2 -15091.59} C_VEL
LIN {X 0,Y 319.608,Z 72.669,A -85,B 0,C 180,E1 -15095.304,E2 -15095.304} C_VEL
LIN {X 0,Y 319.601,Z 72.672,A -85,B 0,C 180,E1 -15098.048,E2 -15098.048} C_VEL
LIN {X 0,Y 319.692,Z 72.661,A -85,B 0,C 180,E1 -15100.962,E2 -15100.962} C_VEL
LIN {X 0,Y 319.734,Z 72.654,A -85,B 0,C 180,E1 -15105.276,E2 -15105.276} C_VEL
LIN {X 0,Y 319.755,Z 72.655,A -85,B 0,C 180,E1 -15109.872,E2 -15109.872} C_VEL
LIN {X 0,Y 319.915,Z 72.633,A -85,B 0,C 180,E1 -15112.425,E2 -15112.425} C_VEL
LIN {X 0,Y 319.746,Z 72.653,A -85,B 0,C 180,E1 -15114.956,E2 -15114.956} C_VEL
LIN {X 0,Y 319.991,Z 72.625,A -85,B 0,C 180,E1 -15117.482,E2 -15117.482} C_VEL
LIN {X 0,Y 320.151,Z 72.605,A -85,B 0,C 180,E1 -15120,E2 -15120} C_VEL
LIN {X 0,Y 319.991,Z 72.623,A -85,B 0,C 180,E1 -15122.517,E2 -15122.517} C_VEL
LIN {X 0,Y 319.938,Z 72.629,A -85,B 0,C 180,E1 -15126.305,E2 -15126.305} C_VEL
LIN {X 0,Y 319.738,Z 72.655,A -85,B 0,C 180,E1 -15130.128,E2 -15130.128} C_VEL
LIN {X 0,Y 319.734,Z 72.654,A -85,B 0,C 180,E1 -15133.992,E2 -15133.992} C_VEL
LIN {X 0,Y 319.66,Z 72.664,A -85,B 0,C 180,E1 -15137.927,E2 -15137.927} C_VEL
LIN {X 0,Y 319.604,Z 72.672,A -85,B 0,C 180,E1 -15140.599,E2 -15140.599} C_VEL
LIN {X 0,Y 319.605,Z 72.674,A -85,B 0,C 180,E1 -15144.696,E2 -15144.696} C_VEL
LIN {X 0,Y 319.617,Z 72.671,A -85,B 0,C 180,E1 -15148.411,E2 -15148.411} C_VEL
LIN {X 0,Y 319.534,Z 72.679,A -85,B 0,C 180,E1 -15151.861,E2 -15151.861} C_VEL
LIN {X 0,Y 319.581,Z 72.674,A -85,B 0,C 180,E1 -15155.543,E2 -15155.543} C_VEL
LIN {X 0,Y 319.559,Z 72.678,A -85,B 0,C 180,E1 -15158.01,E2 -15158.01} C_VEL
LIN {X 0,Y 319.527,Z 72.681,A -85,B 0,C 180,E1 -15161.597,E2 -15161.597} C_VEL
LIN {X 0,Y 319.49,Z 72.684,A -85,B 0,C 180,E1 -15165.257,E2 -15165.257} C_VEL
LIN {X 0,Y 319.53,Z 72.681,A -85,B 0,C 180,E1 -15168.712,E2 -15168.712} C_VEL
LIN {X 0,Y 319.579,Z 72.677,A -85,B 0,C 180,E1 -15172.344,E2 -15172.344} C_VEL
LIN {X 0,Y 319.562,Z 72.678,A -85,B 0,C 180,E1 -15175.123,E2 -15175.123} C_VEL
LIN {X 0,Y 319.596,Z 72.775,A -85,B 0,C 180,E1 -15178.409,E2 -15178.409} C_VEL
LIN {X 0,Y 322.459,Z 86.397,A -85,B 0,C 180,E1 -15182.057,E2 -15182.057} C_VEL
LIN {X 0,Y 323.339,Z 92.304,A -85,B 0,C 180,E1 -15183.571,E2 -15183.571} C_VEL
LIN {X 0,Y 321.966,Z 105.077,A -85,B 0,C 180,E1 -15186.616,E2 -15186.616} C_VEL
LIN {X 0,Y 327.252,Z 147.277,A -85,B 0,C 180,E1 -15187.895,E2 -15187.895} C_VEL
LIN {X 0,Y 326.118,Z 213.809,A -85,B 0,C 180,E1 -15189.377,E2 -15189.377} C_VEL
LIN {X 0,Y 325.409,Z 227.17,A -85,B 0,C 180,E1 -15189.907,E2 -15189.907} C_VEL
LIN {X 0,Y 324.536,Z 239.422,A -85,B 0,C 180,E1 -15190.634,E2 -15190.634} C_VEL
LIN {X 0,Y 323.351,Z 251.755,A -85,B 0,C 180,E1 -15191.629,E2 -15191.629} C_VEL
LIN {X 0,Y 322.245,Z 262.118,A -85,B 0,C 180,E1 -15192.713,E2 -15192.713} C_VEL
LIN {X 0,Y 321.153,Z 273.31,A -85,B 0,C 180,E1 -15194.189,E2 -15194.189} C_VEL
LIN {X 0,Y 320.259,Z 282.562,A -85,B 0,C 180,E1 -15195.707,E2 -15195.707} C_VEL
LIN {X 0,Y 319.4,Z 290.465,A -85,B 0,C 180,E1 -15197.288,E2 -15197.288} C_VEL
LIN {X 0,Y 318.582,Z 298.165,A -85,B 0,C 180,E1 -15199.192,E2 -15199.192} C_VEL
LIN {X 0,Y 318.188,Z 304.364,A -85,B 0,C 180,E1 -15201.105,E2 -15201.105} C_VEL
LIN {X 0,Y 317.965,Z 309.263,A -85,B 0,C 180,E1 -15203.017,E2 -15203.017} C_VEL
LIN {X 0,Y 317.907,Z 313.01,A -85,B 0,C 180,E1 -15204.926,E2 -15204.926} C_VEL
LIN {X 0,Y 317.944,Z 314.938,A -85,B 0,C 180,E1 -15206.197,E2 -15206.197} C_VEL
LIN {X 0,Y 317.942,Z 316.412,A -85,B 0,C 180,E1 -15207.466,E2 -15207.466} C_VEL
LIN {X 0,Y 318.057,Z 317.446,A -85,B 0,C 180,E1 -15208.733,E2 -15208.733} C_VEL
LIN {X 0,Y 318.114,Z 318.078,A -85,B 0,C 180,E1 -15210,E2 -15210} C_VEL
LIN {X 0,Y 317.967,Z 318.307,A -85,B 0,C 180,E1 -15211.266,E2 -15211.266} C_VEL
LIN {X 0,Y 317.867,Z 318.131,A -85,B 0,C 180,E1 -15212.534,E2 -15212.534} C_VEL
LIN {X 0,Y 317.879,Z 317.532,A -85,B 0,C 180,E1 -15213.803,E2 -15213.803} C_VEL
LIN {X 0,Y 317.88,Z 315.162,A -85,B 0,C 180,E1 -15216.346,E2 -15216.346} C_VEL
LIN {X 0,Y 318.141,Z 312.277,A -85,B 0,C 180,E1 -15218.255,E2 -15218.255} C_VEL
LIN {X 0,Y 318.583,Z 308.383,A -85,B 0,C 180,E1 -15220.164,E2 -15220.164} C_VEL
LIN {X 0,Y 319.372,Z 303.387,A -85,B 0,C 180,E1 -15222.066,E2 -15222.066} C_VEL
LIN {X 0,Y 320.626,Z 297.143,A -85,B 0,C 180,E1 -15223.952,E2 -15223.952} C_VEL
LIN {X 0,Y 321.904,Z 289.789,A -85,B 0,C 180,E1 -15225.749,E2 -15225.749} C_VEL
LIN {X 0,Y 323.352,Z 281.689,A -85,B 0,C 180,E1 -15227.356,E2 -15227.356} C_VEL
LIN {X 0,Y 325.203,Z 271.921,A -85,B 0,C 180,E1 -15228.915,E2 -15228.915} C_VEL
LIN {X 0,Y 326.965,Z 261.317,A -85,B 0,C 180,E1 -15230.279,E2 -15230.279} C_VEL
LIN {X 0,Y 328.64,Z 251.091,A -85,B 0,C 180,E1 -15231.318,E2 -15231.318} C_VEL
LIN {X 0,Y 330.288,Z 238.99,A -85,B 0,C 180,E1 -15232.273,E2 -15232.273} C_VEL
LIN {X 0,Y 331.706,Z 225.58,A -85,B 0,C 180,E1 -15233.035,E2 -15233.035} C_VEL
LIN {X 0,Y 332.621,Z 213.21,A -85,B 0,C 180,E1 -15233.503,E2 -15233.503} C_VEL
LIN {X 0,Y 334.252,Z 149.82,A -85,B 0,C 180,E1 -15234.922,E2 -15234.922} C_VEL
LIN {X 0,Y 331.245,Z 130.577,A -85,B 0,C 180,E1 -15235.686,E2 -15235.686} C_VEL
LIN {X 0,Y 326.633,Z 108.133,A -85,B 0,C 180,E1 -15236.717,E2 -15236.717} C_VEL
LIN {X 0,Y 325.749,Z 103.862,A -85,B 0,C 180,E1 -15236.94,E2 -15236.94} C_VEL
LIN {X 0,Y 326.023,Z 100.151,A -85,B 0,C 180,E1 -15237.892,E2 -15237.892} C_VEL
LIN {X 0,Y 324.05,Z 90.685,A -85,B 0,C 180,E1 -15240.64,E2 -15240.64} C_VEL
LIN {X 0,Y 321.861,Z 81.268,A -85,B 0,C 180,E1 -15243.537,E2 -15243.537} C_VEL
LIN {X 0,Y 319.592,Z 72.679,A -85,B 0,C 180,E1 -15246.423,E2 -15246.423} C_VEL
LIN {X 0,Y 319.557,Z 72.681,A -85,B 0,C 180,E1 -15249.668,E2 -15249.668} C_VEL
LIN {X 0,Y 319.544,Z 72.683,A -85,B 0,C 180,E1 -15253.465,E2 -15253.465} C_VEL
LIN {X 0,Y 319.573,Z 72.671,A -85,B 0,C 180,E1 -15257.02,E2 -15257.02} C_VEL
LIN {X 0,Y 319.579,Z 72.675,A -85,B 0,C 180,E1 -15260.376,E2 -15260.376} C_VEL
LIN {X 0,Y 319.558,Z 72.68,A -85,B 0,C 180,E1 -15263.572,E2 -15263.572} C_VEL
LIN {X 0,Y 319.575,Z 72.674,A -85,B 0,C 180,E1 -15266.686,E2 -15266.686} C_VEL
LIN {X 0,Y 319.589,Z 72.669,A -85,B 0,C 180,E1 -15269.616,E2 -15269.616} C_VEL
LIN {X 0,Y 319.606,Z 72.669,A -85,B 0,C 180,E1 -15272.498,E2 -15272.498} C_VEL
LIN {X 0,Y 319.603,Z 72.674,A -85,B 0,C 180,E1 -15275.304,E2 -15275.304} C_VEL
LIN {X 0,Y 319.619,Z 72.67,A -85,B 0,C 180,E1 -15279.402,E2 -15279.402} C_VEL
LIN {X 0,Y 319.656,Z 72.657,A -85,B 0,C 180,E1 -15282.073,E2 -15282.073} C_VEL
LIN {X 0,Y 319.729,Z 72.653,A -85,B 0,C 180,E1 -15286.008,E2 -15286.008} C_VEL
LIN {X 0,Y 319.755,Z 72.656,A -85,B 0,C 180,E1 -15289.873,E2 -15289.873} C_VEL
LIN {X 0,Y 319.922,Z 72.622,A -85,B 0,C 180,E1 -15292.426,E2 -15292.426} C_VEL
LIN {X 0,Y 319.742,Z 72.655,A -85,B 0,C 180,E1 -15294.956,E2 -15294.956} C_VEL
LIN {X 0,Y 319.987,Z 72.615,A -85,B 0,C 180,E1 -15297.483,E2 -15297.483} C_VEL
LIN {X 0,Y 320.146,Z 72.608,A -85,B 0,C 180,E1 -15300,E2 -15300} C_VEL
LIN {X 0,Y 319.986,Z 72.614,A -85,B 0,C 180,E1 -15302.518,E2 -15302.518} C_VEL
LIN {X 0,Y 319.911,Z 72.629,A -85,B 0,C 180,E1 -15306.58,E2 -15306.58} C_VEL
LIN {X 0,Y 319.733,Z 72.657,A -85,B 0,C 180,E1 -15310.128,E2 -15310.128} C_VEL
LIN {X 0,Y 319.73,Z 72.654,A -85,B 0,C 180,E1 -15313.993,E2 -15313.993} C_VEL
LIN {X 0,Y 319.622,Z 72.662,A -85,B 0,C 180,E1 -15317.929,E2 -15317.929} C_VEL
LIN {X 0,Y 319.586,Z 72.674,A -85,B 0,C 180,E1 -15320.601,E2 -15320.601} C_VEL
LIN {X 0,Y 319.556,Z 72.68,A -85,B 0,C 180,E1 -15323.321,E2 -15323.321} C_VEL
LIN {X 0,Y 319.577,Z 72.669,A -85,B 0,C 180,E1 -15326.094,E2 -15326.094} C_VEL
LIN {X 0,Y 319.556,Z 72.674,A -85,B 0,C 180,E1 -15328.937,E2 -15328.937} C_VEL
LIN {X 0,Y 319.523,Z 72.682,A -85,B 0,C 180,E1 -15331.863,E2 -15331.863} C_VEL
LIN {X 0,Y 319.578,Z 72.672,A -85,B 0,C 180,E1 -15335.543,E2 -15335.543} C_VEL
LIN {X 0,Y 319.558,Z 72.681,A -85,B 0,C 180,E1 -15339.669,E2 -15339.669} C_VEL
LIN {X 0,Y 319.52,Z 72.693,A -85,B 0,C 180,E1 -15343.461,E2 -15343.461} C_VEL
LIN {X 0,Y 319.565,Z 72.834,A -85,B 0,C 180,E1 -15347.737,E2 -15347.737} C_VEL
LIN {X 0,Y 320.107,Z 74.917,A -85,B 0,C 180,E1 -15348.495,E2 -15348.495} C_VEL
LIN {X 0,Y 330.268,Z 95.297,A -85,B 0,C 180,E1 -15350.124,E2 -15350.124} C_VEL
LIN {X 0,Y 335.452,Z 107.244,A -85,B 0,C 180,E1 -15350.941,E2 -15350.941} C_VEL
LIN {X 0,Y 333.453,Z 180.513,A -85,B 0,C 180,E1 -15352.561,E2 -15352.561} C_VEL
LIN {X 0,Y 332.655,Z 193.827,A -85,B 0,C 180,E1 -15353.084,E2 -15353.084} C_VEL
LIN {X 0,Y 331.692,Z 206.555,A -85,B 0,C 180,E1 -15353.848,E2 -15353.848} C_VEL
LIN {X 0,Y 330.44,Z 217.977,A -85,B 0,C 180,E1 -15354.767,E2 -15354.767} C_VEL
LIN {X 0,Y 328.972,Z 228.776,A -85,B 0,C 180,E1 -15355.89,E2 -15355.89} C_VEL
LIN {X 0,Y 327.258,Z 239.519,A -85,B 0,C 180,E1 -15357.297,E2 -15357.297} C_VEL
LIN {X 0,Y 325.56,Z 248.746,A -85,B 0,C 180,E1 -15358.796,E2 -15358.796} C_VEL
LIN {X 0,Y 324.056,Z 256.882,A -85,B 0,C 180,E1 -15360.437,E2 -15360.437} C_VEL
LIN {X 0,Y 322.43,Z 264.702,A -85,B 0,C 180,E1 -15362.408,E2 -15362.408} C_VEL
LIN {X 0,Y 321.271,Z 269.972,A -85,B 0,C 180,E1 -15364.055,E2 -15364.055} C_VEL
LIN {X 0,Y 320.178,Z 275.008,A -85,B 0,C 180,E1 -15366.042,E2 -15366.042} C_VEL
LIN {X 0,Y 319.373,Z 278.82,A -85,B 0,C 180,E1 -15368.032,E2 -15368.032} C_VEL
LIN {X 0,Y 318.903,Z 280.759,A -85,B 0,C 180,E1 -15369.354,E2 -15369.354} C_VEL
LIN {X 0,Y 318.293,Z 283.044,A -85,B 0,C 180,E1 -15371.707,E2 -15371.707} C_VEL
LIN {X 0,Y 318.04,Z 283.81,A -85,B 0,C 180,E1 -15373.306,E2 -15373.306} C_VEL
LIN {X 0,Y 317.901,Z 283.992,A -85,B 0,C 180,E1 -15374.616,E2 -15374.616} C_VEL
LIN {X 0,Y 317.91,Z 283.452,A -85,B 0,C 180,E1 -15376.584,E2 -15376.584} C_VEL
LIN {X 0,Y 317.928,Z 281.987,A -85,B 0,C 180,E1 -15378.525,E2 -15378.525} C_VEL
LIN {X 0,Y 318.05,Z 280.477,A -85,B 0,C 180,E1 -15379.818,E2 -15379.818} C_VEL
LIN {X 0,Y 318.348,Z 277.399,A -85,B 0,C 180,E1 -15381.75,E2 -15381.75} C_VEL
LIN {X 0,Y 318.764,Z 273.26,A -85,B 0,C 180,E1 -15383.671,E2 -15383.671} C_VEL
LIN {X 0,Y 319.315,Z 266.949,A -85,B 0,C 180,E1 -15385.899,E2 -15385.899} C_VEL
LIN {X 0,Y 320.044,Z 260.081,A -85,B 0,C 180,E1 -15387.798,E2 -15387.798} C_VEL
LIN {X 0,Y 320.89,Z 253.055,A -85,B 0,C 180,E1 -15389.373,E2 -15389.373} C_VEL
LIN {X 0,Y 321.891,Z 244.588,A -85,B 0,C 180,E1 -15390.939,E2 -15390.939} C_VEL
LIN {X 0,Y 323.004,Z 234.135,A -85,B 0,C 180,E1 -15392.495,E2 -15392.495} C_VEL
LIN {X 0,Y 324.14,Z 222.774,A -85,B 0,C 180,E1 -15393.84,E2 -15393.84} C_VEL
LIN {X 0,Y 325.107,Z 210.54,A -85,B 0,C 180,E1 -15394.961,E2 -15394.961} C_VEL
LIN {X 0,Y 325.807,Z 198.31,A -85,B 0,C 180,E1 -15395.804,E2 -15395.804} C_VEL
LIN {X 0,Y 326.302,Z 185.9,A -85,B 0,C 180,E1 -15396.412,E2 -15396.412} C_VEL
LIN {X 0,Y 326.694,Z 171.622,A -85,B 0,C 180,E1 -15396.823,E2 -15396.823} C_VEL
LIN {X 0,Y 328.127,Z 98.638,A -85,B 0,C 180,E1 -15398.409,E2 -15398.409} C_VEL
LIN {X 0,Y 322.844,Z 81.442,A -85,B 0,C 180,E1 -15399.123,E2 -15399.123} C_VEL
LIN {X 0,Y 319.943,Z 73.343,A -85,B 0,C 180,E1 -15399.524,E2 -15399.524} C_VEL
LIN {X 0,Y 319.802,Z 72.648,A -85,B 0,C 180,E1 -15399.807,E2 -15399.807} C_VEL
LIN {X 0,Y 319.737,Z 72.658,A -85,B 0,C 180,E1 -15403.992,E2 -15403.992} C_VEL
LIN {X 0,Y 319.663,Z 72.667,A -85,B 0,C 180,E1 -15407.927,E2 -15407.927} C_VEL
LIN {X 0,Y 319.608,Z 72.673,A -85,B 0,C 180,E1 -15410.6,E2 -15410.6} C_VEL
LIN {X 0,Y 319.608,Z 72.672,A -85,B 0,C 180,E1 -15414.696,E2 -15414.696} C_VEL
LIN {X 0,Y 319.615,Z 72.671,A -85,B 0,C 180,E1 -15418.41,E2 -15418.41} C_VEL
LIN {X 0,Y 319.536,Z 72.683,A -85,B 0,C 180,E1 -15421.862,E2 -15421.862} C_VEL
LIN {X 0,Y 319.585,Z 72.676,A -85,B 0,C 180,E1 -15425.543,E2 -15425.543} C_VEL
LIN {X 0,Y 319.535,Z 72.678,A -85,B 0,C 180,E1 -15428.73,E2 -15428.73} C_VEL
LIN {X 0,Y 318.866,Z 72.766,A -85,B 0,C 180,E1 -15429.783,E2 -15429.783} C_VEL
LIN {X 0,Y 316.04,Z 73.12,A -85,B 0,C 180,E1 -15431.498,E2 -15431.498} C_VEL
LIN {X 0,Y 313.63,Z 73.42,A -85,B 0,C 180,E1 -15432.887,E2 -15432.887} C_VEL
LIN {X 0,Y 312.569,Z 73.548,A -85,B 0,C 180,E1 -15433.962,E2 -15433.962} C_VEL
LIN {X 0,Y 312.468,Z 73.558,A -85,B 0,C 180,E1 -15434.326,E2 -15434.326} C_VEL
LIN {X 0,Y 312.49,Z 73.558,A -85,B 0,C 180,E1 -15437.918,E2 -15437.918} C_VEL
LIN {X 0,Y 312.502,Z 73.558,A -85,B 0,C 180,E1 -15440.971,E2 -15440.971} C_VEL
LIN {X 0,Y 312.535,Z 73.543,A -85,B 0,C 180,E1 -15444.22,E2 -15444.22} C_VEL
LIN {X 0,Y 312.507,Z 73.554,A -85,B 0,C 180,E1 -15447.334,E2 -15447.334} C_VEL
LIN {X 0,Y 312.548,Z 73.551,A -85,B 0,C 180,E1 -15451.279,E2 -15451.279} C_VEL
LIN {X 0,Y 312.589,Z 73.547,A -85,B 0,C 180,E1 -15454.711,E2 -15454.711} C_VEL
LIN {X 0,Y 312.591,Z 73.544,A -85,B 0,C 180,E1 -15457.529,E2 -15457.529} C_VEL
LIN {X 0,Y 312.641,Z 73.538,A -85,B 0,C 180,E1 -15461.656,E2 -15461.656} C_VEL
LIN {X 0,Y 312.697,Z 73.531,A -85,B 0,C 180,E1 -15465.686,E2 -15465.686} C_VEL
LIN {X 0,Y 312.701,Z 73.532,A -85,B 0,C 180,E1 -15469.641,E2 -15469.641} C_VEL
LIN {X 0,Y 312.856,Z 73.513,A -85,B 0,C 180,E1 -15472.254,E2 -15472.254} C_VEL
LIN {X 0,Y 312.716,Z 73.529,A -85,B 0,C 180,E1 -15474.842,E2 -15474.842} C_VEL
LIN {X 0,Y 312.991,Z 73.493,A -85,B 0,C 180,E1 -15478.713,E2 -15478.713} C_VEL
LIN {X 0,Y 312.991,Z 73.494,A -85,B 0,C 180,E1 -15481.286,E2 -15481.286} C_VEL
LIN {X 0,Y 312.713,Z 73.531,A -85,B 0,C 180,E1 -15485.157,E2 -15485.157} C_VEL
LIN {X 0,Y 312.894,Z 73.506,A -85,B 0,C 180,E1 -15486.448,E2 -15486.448} C_VEL
LIN {X 0,Y 312.688,Z 73.532,A -85,B 0,C 180,E1 -15490.358,E2 -15490.358} C_VEL
LIN {X 0,Y 312.702,Z 73.532,A -85,B 0,C 180,E1 -15494.887,E2 -15494.887} C_VEL
LIN {X 0,Y 312.631,Z 73.544,A -85,B 0,C 180,E1 -15499.235,E2 -15499.235} C_VEL
LIN {X 0,Y 312.528,Z 73.555,A -85,B 0,C 180,E1 -15502.78,E2 -15502.78} C_VEL
LIN {X 0,Y 312.599,Z 73.543,A -85,B 0,C 180,E1 -15505.933,E2 -15505.933} C_VEL
LIN {X 0,Y 312.547,Z 73.548,A -85,B 0,C 180,E1 -15509.65,E2 -15509.65} C_VEL
LIN {X 0,Y 312.521,Z 73.553,A -85,B 0,C 180,E1 -15513.689,E2 -15513.689} C_VEL
LIN {X 0,Y 312.527,Z 73.553,A -85,B 0,C 180,E1 -15517.385,E2 -15517.385} C_VEL
LIN {X 0,Y 312.491,Z 73.56,A -85,B 0,C 180,E1 -15520.709,E2 -15520.709} C_VEL
LIN {X 0,Y 312.453,Z 73.564,A -85,B 0,C 180,E1 -15524.209,E2 -15524.209} C_VEL
LIN {X 0,Y 312.486,Z 73.562,A -85,B 0,C 180,E1 -15527.918,E2 -15527.918} C_VEL
LIN {X 0,Y 312.536,Z 73.557,A -85,B 0,C 180,E1 -15531.91,E2 -15531.91} C_VEL
LIN {X 0,Y 312.508,Z 73.56,A -85,B 0,C 180,E1 -15535.79,E2 -15535.79} C_VEL
LIN {X 0,Y 312.572,Z 73.753,A -85,B 0,C 180,E1 -15538.109,E2 -15538.109} C_VEL
LIN {X 0,Y 315.368,Z 86.941,A -85,B 0,C 180,E1 -15541.734,E2 -15541.734} C_VEL
LIN {X 0,Y 316.304,Z 92.535,A -85,B 0,C 180,E1 -15543.212,E2 -15543.212} C_VEL
LIN {X 0,Y 315.558,Z 101.177,A -85,B 0,C 180,E1 -15545.333,E2 -15545.333} C_VEL
LIN {X 0,Y 315.17,Z 104.994,A -85,B 0,C 180,E1 -15546.197,E2 -15546.197} C_VEL
LIN {X 0,Y 320.483,Z 147.963,A -85,B 0,C 180,E1 -15547.53,E2 -15547.53} C_VEL
LIN {X 0,Y 319.286,Z 214.128,A -85,B 0,C 180,E1 -15549.041,E2 -15549.041} C_VEL
LIN {X 0,Y 318.503,Z 228.02,A -85,B 0,C 180,E1 -15549.621,E2 -15549.621} C_VEL
LIN {X 0,Y 317.5,Z 240.995,A -85,B 0,C 180,E1 -15550.439,E2 -15550.439} C_VEL
LIN {X 0,Y 316.303,Z 253.627,A -85,B 0,C 180,E1 -15551.541,E2 -15551.541} C_VEL
LIN {X 0,Y 315.155,Z 263.575,A -85,B 0,C 180,E1 -15552.646,E2 -15552.646} C_VEL
LIN {X 0,Y 314.084,Z 274.012,A -85,B 0,C 180,E1 -15554.091,E2 -15554.091} C_VEL
LIN {X 0,Y 313.114,Z 283.358,A -85,B 0,C 180,E1 -15555.705,E2 -15555.705} C_VEL
LIN {X 0,Y 312.266,Z 291.05,A -85,B 0,C 180,E1 -15557.324,E2 -15557.324} C_VEL
LIN {X 0,Y 311.471,Z 298.579,A -85,B 0,C 180,E1 -15559.271,E2 -15559.271} C_VEL
LIN {X 0,Y 311.044,Z 305.518,A -85,B 0,C 180,E1 -15561.554,E2 -15561.554} C_VEL
LIN {X 0,Y 310.827,Z 310.07,A -85,B 0,C 180,E1 -15563.508,E2 -15563.508} C_VEL
LIN {X 0,Y 310.814,Z 312.465,A -85,B 0,C 180,E1 -15564.81,E2 -15564.81} C_VEL
LIN {X 0,Y 310.868,Z 314.421,A -85,B 0,C 180,E1 -15566.111,E2 -15566.111} C_VEL
LIN {X 0,Y 310.855,Z 315.939,A -85,B 0,C 180,E1 -15567.408,E2 -15567.408} C_VEL
LIN {X 0,Y 310.961,Z 317.001,A -85,B 0,C 180,E1 -15568.704,E2 -15568.704} C_VEL
LIN {X 0,Y 311.038,Z 317.658,A -85,B 0,C 180,E1 -15570,E2 -15570} C_VEL
LIN {X 0,Y 310.784,Z 317.771,A -85,B 0,C 180,E1 -15572.592,E2 -15572.592} C_VEL
LIN {X 0,Y 310.781,Z 317.204,A -85,B 0,C 180,E1 -15573.89,E2 -15573.89} C_VEL
LIN {X 0,Y 310.809,Z 314.881,A -85,B 0,C 180,E1 -15576.491,E2 -15576.491} C_VEL
LIN {X 0,Y 311.085,Z 312.045,A -85,B 0,C 180,E1 -15578.444,E2 -15578.444} C_VEL
LIN {X 0,Y 311.568,Z 308.204,A -85,B 0,C 180,E1 -15580.396,E2 -15580.396} C_VEL
LIN {X 0,Y 312.394,Z 303.265,A -85,B 0,C 180,E1 -15582.34,E2 -15582.34} C_VEL
LIN {X 0,Y 313.721,Z 297.084,A -85,B 0,C 180,E1 -15584.265,E2 -15584.265} C_VEL
LIN {X 0,Y 315.019,Z 290.068,A -85,B 0,C 180,E1 -15586.039,E2 -15586.039} C_VEL
LIN {X 0,Y 316.61,Z 281.655,A -85,B 0,C 180,E1 -15587.771,E2 -15587.771} C_VEL
LIN {X 0,Y 318.719,Z 271.118,A -85,B 0,C 180,E1 -15589.482,E2 -15589.482} C_VEL
LIN {X 0,Y 320.636,Z 260.435,A -85,B 0,C 180,E1 -15590.865,E2 -15590.865} C_VEL
LIN {X 0,Y 322.319,Z 250.11,A -85,B 0,C 180,E1 -15591.925,E2 -15591.925} C_VEL
LIN {X 0,Y 324.052,Z 237.764,A -85,B 0,C 180,E1 -15592.893,E2 -15592.893} C_VEL
LIN {X 0,Y 325.461,Z 224.818,A -85,B 0,C 180,E1 -15593.63,E2 -15593.63} C_VEL
LIN {X 0,Y 326.418,Z 212.23,A -85,B 0,C 180,E1 -15594.104,E2 -15594.104} C_VEL
LIN {X 0,Y 328.028,Z 150.524,A -85,B 0,C 180,E1 -15595.509,E2 -15595.509} C_VEL
LIN {X 0,Y 324.789,Z 129.916,A -85,B 0,C 180,E1 -15596.356,E2 -15596.356} C_VEL
LIN {X 0,Y 319.708,Z 105.777,A -85,B 0,C 180,E1 -15597.525,E2 -15597.525} C_VEL
LIN {X 0,Y 319.248,Z 103.366,A -85,B 0,C 180,E1 -15597.677,E2 -15597.677} C_VEL
LIN {X 0,Y 318.604,Z 98.622,A -85,B 0,C 180,E1 -15599.031,E2 -15599.031} C_VEL
LIN {X 0,Y 315.982,Z 86.85,A -85,B 0,C 180,E1 -15602.639,E2 -15602.639} C_VEL
LIN {X 0,Y 313.259,Z 76.292,A -85,B 0,C 180,E1 -15606.132,E2 -15606.132} C_VEL
LIN {X 0,Y 312.537,Z 73.554,A -85,B 0,C 180,E1 -15607.108,E2 -15607.108} C_VEL
LIN {X 0,Y 312.488,Z 73.56,A -85,B 0,C 180,E1 -15610.709,E2 -15610.709} C_VEL
LIN {X 0,Y 312.457,Z 73.557,A -85,B 0,C 180,E1 -15614.208,E2 -15614.208} C_VEL
LIN {X 0,Y 312.525,Z 73.557,A -85,B 0,C 180,E1 -15617.909,E2 -15617.909} C_VEL
LIN {X 0,Y 312.541,Z 73.548,A -85,B 0,C 180,E1 -15621.908,E2 -15621.908} C_VEL
LIN {X 0,Y 312.504,Z 73.551,A -85,B 0,C 180,E1 -15625.79,E2 -15625.79} C_VEL
LIN {X 0,Y 312.521,Z 73.55,A -85,B 0,C 180,E1 -15628.854,E2 -15628.854} C_VEL
LIN {X 0,Y 312.572,Z 73.548,A -85,B 0,C 180,E1 -15631.825,E2 -15631.825} C_VEL
LIN {X 0,Y 312.583,Z 73.546,A -85,B 0,C 180,E1 -15634.711,E2 -15634.711} C_VEL
LIN {X 0,Y 312.585,Z 73.536,A -85,B 0,C 180,E1 -15637.529,E2 -15637.529} C_VEL
LIN {X 0,Y 312.636,Z 73.533,A -85,B 0,C 180,E1 -15641.656,E2 -15641.656} C_VEL
LIN {X 0,Y 312.691,Z 73.534,A -85,B 0,C 180,E1 -15645.686,E2 -15645.686} C_VEL
LIN {X 0,Y 312.699,Z 73.533,A -85,B 0,C 180,E1 -15649.642,E2 -15649.642} C_VEL
LIN {X 0,Y 312.863,Z 73.501,A -85,B 0,C 180,E1 -15652.254,E2 -15652.254} C_VEL
LIN {X 0,Y 312.713,Z 73.531,A -85,B 0,C 180,E1 -15654.843,E2 -15654.843} C_VEL
LIN {X 0,Y 312.988,Z 73.492,A -85,B 0,C 180,E1 -15658.714,E2 -15658.714} C_VEL
LIN {X 0,Y 312.986,Z 73.496,A -85,B 0,C 180,E1 -15661.287,E2 -15661.287} C_VEL
LIN {X 0,Y 312.71,Z 73.532,A -85,B 0,C 180,E1 -15665.158,E2 -15665.158} C_VEL
LIN {X 0,Y 312.878,Z 73.507,A -85,B 0,C 180,E1 -15666.557,E2 -15666.557} C_VEL
LIN {X 0,Y 312.683,Z 73.535,A -85,B 0,C 180,E1 -15670.359,E2 -15670.359} C_VEL
LIN {X 0,Y 312.665,Z 73.537,A -85,B 0,C 180,E1 -15674.866,E2 -15674.866} C_VEL
LIN {X 0,Y 312.586,Z 73.549,A -85,B 0,C 180,E1 -15679.215,E2 -15679.215} C_VEL
LIN {X 0,Y 312.523,Z 73.55,A -85,B 0,C 180,E1 -15682.781,E2 -15682.781} C_VEL
LIN {X 0,Y 312.536,Z 73.545,A -85,B 0,C 180,E1 -15685.912,E2 -15685.912} C_VEL
LIN {X 0,Y 312.502,Z 73.552,A -85,B 0,C 180,E1 -15689.655,E2 -15689.655} C_VEL
LIN {X 0,Y 312.518,Z 73.556,A -85,B 0,C 180,E1 -15693.69,E2 -15693.69} C_VEL
LIN {X 0,Y 312.514,Z 73.557,A -85,B 0,C 180,E1 -15697.387,E2 -15697.387} C_VEL
LIN {X 0,Y 312.487,Z 73.55,A -85,B 0,C 180,E1 -15700.71,E2 -15700.71} C_VEL
LIN {X 0,Y 312.451,Z 73.564,A -85,B 0,C 180,E1 -15704.211,E2 -15704.211} C_VEL
LIN {X 0,Y 312.516,Z 73.604,A -85,B 0,C 180,E1 -15707.013,E2 -15707.013} C_VEL
LIN {X 0,Y 312.962,Z 75.434,A -85,B 0,C 180,E1 -15707.669,E2 -15707.669} C_VEL
LIN {X 0,Y 322.452,Z 93.891,A -85,B 0,C 180,E1 -15709.255,E2 -15709.255} C_VEL
LIN {X 0,Y 329.285,Z 109.133,A -85,B 0,C 180,E1 -15710.369,E2 -15710.369} C_VEL
LIN {X 0,Y 327.166,Z 181.7,A -85,B 0,C 180,E1 -15712.007,E2 -15712.007} C_VEL
LIN {X 0,Y 326.308,Z 195.375,A -85,B 0,C 180,E1 -15712.572,E2 -15712.572} C_VEL
LIN {X 0,Y 325.318,Z 207.561,A -85,B 0,C 180,E1 -15713.332,E2 -15713.332} C_VEL
LIN {X 0,Y 323.906,Z 219.468,A -85,B 0,C 180,E1 -15714.33,E2 -15714.33} C_VEL
LIN {X 0,Y 322.404,Z 230.062,A -85,B 0,C 180,E1 -15715.476,E2 -15715.476} C_VEL
LIN {X 0,Y 320.546,Z 240.945,A -85,B 0,C 180,E1 -15716.95,E2 -15716.95} C_VEL
LIN {X 0,Y 318.843,Z 249.732,A -85,B 0,C 180,E1 -15718.433,E2 -15718.433} C_VEL
LIN {X 0,Y 317.184,Z 258.048,A -85,B 0,C 180,E1 -15720.18,E2 -15720.18} C_VEL
LIN {X 0,Y 315.576,Z 265.461,A -85,B 0,C 180,E1 -15722.117,E2 -15722.117} C_VEL
LIN {X 0,Y 314.151,Z 271.589,A -85,B 0,C 180,E1 -15724.136,E2 -15724.136} C_VEL
LIN {X 0,Y 313.077,Z 276.356,A -85,B 0,C 180,E1 -15726.168,E2 -15726.168} C_VEL
LIN {X 0,Y 312.233,Z 279.919,A -85,B 0,C 180,E1 -15728.199,E2 -15728.199} C_VEL
LIN {X 0,Y 311.587,Z 282.394,A -85,B 0,C 180,E1 -15730.225,E2 -15730.225} C_VEL
LIN {X 0,Y 311.248,Z 283.467,A -85,B 0,C 180,E1 -15731.572,E2 -15731.572} C_VEL
LIN {X 0,Y 311.009,Z 284.119,A -85,B 0,C 180,E1 -15732.917,E2 -15732.917} C_VEL
LIN {X 0,Y 310.854,Z 284.369,A -85,B 0,C 180,E1 -15734.259,E2 -15734.259} C_VEL
LIN {X 0,Y 310.813,Z 283.846,A -85,B 0,C 180,E1 -15736.486,E2 -15736.486} C_VEL
LIN {X 0,Y 310.839,Z 282.57,A -85,B 0,C 180,E1 -15738.26,E2 -15738.26} C_VEL
LIN {X 0,Y 310.924,Z 281.162,A -85,B 0,C 180,E1 -15739.582,E2 -15739.582} C_VEL
LIN {X 0,Y 311.229,Z 278.192,A -85,B 0,C 180,E1 -15741.56,E2 -15741.56} C_VEL
LIN {X 0,Y 311.643,Z 274.181,A -85,B 0,C 180,E1 -15743.526,E2 -15743.526} C_VEL
LIN {X 0,Y 312.191,Z 268.025,A -85,B 0,C 180,E1 -15745.805,E2 -15745.805} C_VEL
LIN {X 0,Y 312.926,Z 261.306,A -85,B 0,C 180,E1 -15747.748,E2 -15747.748} C_VEL
LIN {X 0,Y 313.971,Z 252.956,A -85,B 0,C 180,E1 -15749.68,E2 -15749.68} C_VEL
LIN {X 0,Y 315.013,Z 244.355,A -85,B 0,C 180,E1 -15751.279,E2 -15751.279} C_VEL
LIN {X 0,Y 316.204,Z 233.534,A -85,B 0,C 180,E1 -15752.899,E2 -15752.899} C_VEL
LIN {X 0,Y 317.38,Z 222.037,A -85,B 0,C 180,E1 -15754.259,E2 -15754.259} C_VEL
LIN {X 0,Y 318.319,Z 209.684,A -85,B 0,C 180,E1 -15755.385,E2 -15755.385} C_VEL
LIN {X 0,Y 319.041,Z 197.078,A -85,B 0,C 180,E1 -15756.245,E2 -15756.245} C_VEL
LIN {X 0,Y 319.6,Z 184.568,A -85,B 0,C 180,E1 -15756.828,E2 -15756.828} C_VEL
LIN {X 0,Y 320.034,Z 167.045,A -85,B 0,C 180,E1 -15757.294,E2 -15757.294} C_VEL
LIN {X 0,Y 321.308,Z 99.304,A -85,B 0,C 180,E1 -15758.8,E2 -15758.8} C_VEL
LIN {X 0,Y 315.573,Z 81.426,A -85,B 0,C 180,E1 -15759.584,E2 -15759.584} C_VEL
LIN {X 0,Y 312.779,Z 73.723,A -85,B 0,C 180,E1 -15759.978,E2 -15759.978} C_VEL
LIN {X 0,Y 312.699,Z 73.538,A -85,B 0,C 180,E1 -15764.314,E2 -15764.314} C_VEL
LIN {X 0,Y 312.643,Z 73.543,A -85,B 0,C 180,E1 -15768.344,E2 -15768.344} C_VEL
LIN {X 0,Y 312.531,Z 73.552,A -85,B 0,C 180,E1 -15772.781,E2 -15772.781} C_VEL
LIN {X 0,Y 312.607,Z 73.547,A -85,B 0,C 180,E1 -15775.936,E2 -15775.936} C_VEL
LIN {X 0,Y 312.543,Z 73.553,A -85,B 0,C 180,E1 -15779.651,E2 -15779.651} C_VEL
LIN {X 0,Y 312.524,Z 73.554,A -85,B 0,C 180,E1 -15783.689,E2 -15783.689} C_VEL
LIN {X 0,Y 312.543,Z 73.553,A -85,B 0,C 180,E1 -15787.383,E2 -15787.383} C_VEL
LIN {X 0,Y 312.494,Z 73.556,A -85,B 0,C 180,E1 -15790.709,E2 -15790.709} C_VEL
LIN {X 0,Y 312.468,Z 73.558,A -85,B 0,C 180,E1 -15794.326,E2 -15794.326} C_VEL
LIN {X 0,Y 311.777,Z 73.649,A -85,B 0,C 180,E1 -15795.402,E2 -15795.402} C_VEL
LIN {X 0,Y 308.974,Z 73.998,A -85,B 0,C 180,E1 -15797.156,E2 -15797.156} C_VEL
LIN {X 0,Y 306.599,Z 74.296,A -85,B 0,C 180,E1 -15798.578,E2 -15798.578} C_VEL
LIN {X 0,Y 305.552,Z 74.422,A -85,B 0,C 180,E1 -15799.677,E2 -15799.677} C_VEL
LIN {X 0,Y 305.449,Z 74.432,A -85,B 0,C 180,E1 -15800.05,E2 -15800.05} C_VEL
LIN {X 0,Y 305.484,Z 74.421,A -85,B 0,C 180,E1 -15803.632,E2 -15803.632} C_VEL
LIN {X 0,Y 305.468,Z 74.426,A -85,B 0,C 180,E1 -15806.483,E2 -15806.483} C_VEL
LIN {X 0,Y 305.461,Z 74.432,A -85,B 0,C 180,E1 -15809.59,E2 -15809.59} C_VEL
LIN {X 0,Y 305.518,Z 74.43,A -85,B 0,C 180,E1 -15812.608,E2 -15812.608} C_VEL
LIN {X 0,Y 305.511,Z 74.423,A -85,B 0,C 180,E1 -15815.539,E2 -15815.539} C_VEL
LIN {X 0,Y 305.523,Z 74.426,A -85,B 0,C 180,E1 -15819.815,E2 -15819.815} C_VEL
LIN {X 0,Y 305.577,Z 74.419,A -85,B 0,C 180,E1 -15822.603,E2 -15822.603} C_VEL
LIN {X 0,Y 305.652,Z 74.408,A -85,B 0,C 180,E1 -15825.349,E2 -15825.349} C_VEL
LIN {X 0,Y 305.638,Z 74.41,A -85,B 0,C 180,E1 -15829.399,E2 -15829.399} C_VEL
LIN {X 0,Y 305.8,Z 74.392,A -85,B 0,C 180,E1 -15832.074,E2 -15832.074} C_VEL
LIN {X 0,Y 305.688,Z 74.404,A -85,B 0,C 180,E1 -15834.723,E2 -15834.723} C_VEL
LIN {X 0,Y 305.958,Z 74.369,A -85,B 0,C 180,E1 -15838.683,E2 -15838.683} C_VEL
LIN {X 0,Y 305.958,Z 74.37,A -85,B 0,C 180,E1 -15841.316,E2 -15841.316} C_VEL
LIN {X 0,Y 305.684,Z 74.407,A -85,B 0,C 180,E1 -15845.276,E2 -15845.276} C_VEL
LIN {X 0,Y 305.773,Z 74.393,A -85,B 0,C 180,E1 -15847.926,E2 -15847.926} C_VEL
LIN {X 0,Y 305.601,Z 74.416,A -85,B 0,C 180,E1 -15851.945,E2 -15851.945} C_VEL
LIN {X 0,Y 305.64,Z 74.413,A -85,B 0,C 180,E1 -15855.035,E2 -15855.035} C_VEL
LIN {X 0,Y 305.577,Z 74.421,A -85,B 0,C 180,E1 -15859.444,E2 -15859.444} C_VEL
LIN {X 0,Y 305.488,Z 74.434,A -85,B 0,C 180,E1 -15863.039,E2 -15863.039} C_VEL
LIN {X 0,Y 305.528,Z 74.424,A -85,B 0,C 180,E1 -15866.219,E2 -15866.219} C_VEL
LIN {X 0,Y 305.497,Z 74.429,A -85,B 0,C 180,E1 -15869.05,E2 -15869.05} C_VEL
LIN {X 0,Y 305.466,Z 74.432,A -85,B 0,C 180,E1 -15873.516,E2 -15873.516} C_VEL
LIN {X 0,Y 305.476,Z 74.434,A -85,B 0,C 180,E1 -15876.739,E2 -15876.739} C_VEL
LIN {X 0,Y 305.456,Z 74.437,A -85,B 0,C 180,E1 -15880.599,E2 -15880.599} C_VEL
LIN {X 0,Y 305.427,Z 74.437,A -85,B 0,C 180,E1 -15883.655,E2 -15883.655} C_VEL
LIN {X 0,Y 305.456,Z 74.434,A -85,B 0,C 180,E1 -15887.414,E2 -15887.414} C_VEL
LIN {X 0,Y 305.496,Z 74.432,A -85,B 0,C 180,E1 -15891.6,E2 -15891.6} C_VEL
LIN {X 0,Y 305.464,Z 74.434,A -85,B 0,C 180,E1 -15894.887,E2 -15894.887} C_VEL
LIN {X 0,Y 305.511,Z 74.613,A -85,B 0,C 180,E1 -15897.764,E2 -15897.764} C_VEL
LIN {X 0,Y 308.285,Z 87.481,A -85,B 0,C 180,E1 -15901.396,E2 -15901.396} C_VEL
LIN {X 0,Y 309.355,Z 94.708,A -85,B 0,C 180,E1 -15903.34,E2 -15903.34} C_VEL
LIN {X 0,Y 308.268,Z 104.29,A -85,B 0,C 180,E1 -15905.729,E2 -15905.729} C_VEL
LIN {X 0,Y 313.551,Z 147.214,A -85,B 0,C 180,E1 -15907.106,E2 -15907.106} C_VEL
LIN {X 0,Y 313.697,Z 154.665,A -85,B 0,C 180,E1 -15907.292,E2 -15907.292} C_VEL
LIN {X 0,Y 312.503,Z 213.268,A -85,B 0,C 180,E1 -15908.651,E2 -15908.651} C_VEL
LIN {X 0,Y 311.783,Z 226.567,A -85,B 0,C 180,E1 -15909.205,E2 -15909.205} C_VEL
LIN {X 0,Y 310.824,Z 239.356,A -85,B 0,C 180,E1 -15910.001,E2 -15910.001} C_VEL
LIN {X 0,Y 309.665,Z 250.685,A -85,B 0,C 180,E1 -15910.958,E2 -15910.958} C_VEL
LIN {X 0,Y 308.435,Z 261.096,A -85,B 0,C 180,E1 -15912.084,E2 -15912.084} C_VEL
LIN {X 0,Y 307.327,Z 271.9,A -85,B 0,C 180,E1 -15913.561,E2 -15913.561} C_VEL
LIN {X 0,Y 306.469,Z 279.563,A -85,B 0,C 180,E1 -15914.833,E2 -15914.833} C_VEL
LIN {X 0,Y 305.453,Z 288.813,A -85,B 0,C 180,E1 -15916.697,E2 -15916.697} C_VEL
LIN {X 0,Y 304.531,Z 296.72,A -85,B 0,C 180,E1 -15918.687,E2 -15918.687} C_VEL
LIN {X 0,Y 304.069,Z 303.048,A -85,B 0,C 180,E1 -15920.689,E2 -15920.689} C_VEL
LIN {X 0,Y 303.814,Z 308.064,A -85,B 0,C 180,E1 -15922.69,E2 -15922.69} C_VEL
LIN {X 0,Y 303.717,Z 311.92,A -85,B 0,C 180,E1 -15924.689,E2 -15924.689} C_VEL
LIN {X 0,Y 303.794,Z 313.903,A -85,B 0,C 180,E1 -15926.02,E2 -15926.02} C_VEL
LIN {X 0,Y 303.772,Z 315.454,A -85,B 0,C 180,E1 -15927.347,E2 -15927.347} C_VEL
LIN {X 0,Y 303.866,Z 316.556,A -85,B 0,C 180,E1 -15928.674,E2 -15928.674} C_VEL
LIN {X 0,Y 303.948,Z 317.237,A -85,B 0,C 180,E1 -15930,E2 -15930} C_VEL
LIN {X 0,Y 303.702,Z 317.401,A -85,B 0,C 180,E1 -15932.652,E2 -15932.652} C_VEL
LIN {X 0,Y 303.686,Z 316.876,A -85,B 0,C 180,E1 -15933.981,E2 -15933.981} C_VEL
